C01743=-16.662,-86.143,37.169,176.3239,-5.7975,-6670.9471
C01744=-18.041,-88.518,38.031,179.9182,-0.1571,-6671.5198
C01745=-19.458,-91.164,38.697,-178.4928,2.5231,-6672.0484
C01746=-21.221,-93.510,39.027,-177.6909,1.9849,-6672.7860
C01747=-24.227,-95.023,39.203,-178.2776,0.4750,-6674.3034
C01748=-28.112,-95.435,39.346,-178.7289,-0.0594,-6676.4132
C01749=-32.220,-94.603,39.491,-179.9530,-0.0151,-6678.8079
C01750=-36.266,-93.184,39.587,-179.9934,-0.0025,-6681.2653
C01751=-40.247,-91.535,39.587,-179.9935,-0.0029,-6683.7346
C01752=-44.111,-89.678,39.491,-179.9560,-0.0226,-6686.1917
C01753=-47.604,-87.360,39.346,-179.0591,-0.8569,-6688.5867
C01754=-50.060,-84.322,39.203,-179.1177,-1.5538,-6690.6966
C01755=-51.116,-81.128,39.027,-179.7705,-3.0349,-6692.2136
C01756=-50.704,-78.221,38.697,179.2808,-2.8489,-6692.9519
C01757=-49.835,-75.348,38.031,-179.9468,0.1689,-6693.4806
C01758=-49.130,-72.694,37.169,-178.4898,6.6859,-6694.0527
C01759=-49.058,-70.314,36.333,179.0727,19.5923,-6694.9034
C01760=-50.194,-67.954,35.726,158.7492,29.2297,-6696.4513
C01761=-53.078,-65.141,35.484,150.6424,26.8233,-6699.1737
C01762=-56.256,-62.380,35.473,150.4564,26.9203,-6702.0450
C01763=-59.399,-59.399,35.480,151.7261,28.2744,-6705.0000
C01764=-62.380,-56.256,35.473,153.0793,29.5434,-6707.9550
C01765=-65.141,-53.078,35.484,153.1760,29.3567,-6710.8263
C01766=-67.954,-50.194,35.726,150.7705,21.2516,-6713.5487
C01767=-70.314,-49.058,36.333,160.4077,0.9273,-6715.0966
C01768=-72.694,-49.130,37.169,173.3141,-1.5102,-6715.9473
C01769=-75.348,-49.835,38.031,179.8311,-0.0532,-6716.5194
C01770=-78.221,-50.704,38.697,-177.1511,0.7192,-6717.0481
C01771=-81.128,-51.116,39.027,-176.9651,-0.2295,-6717.7864
C01772=-84.322,-50.060,39.203,-178.4462,-0.8823,-6719.3034
C01773=-87.360,-47.604,39.346,-179.1431,-0.9409,-6721.4133
C01774=-89.678,-44.111,39.491,-179.9774,-0.0440,-6723.8083
C01775=-91.535,-40.247,39.587,-179.9971,-0.0065,-6726.2654
C01776=-93.184,-36.266,39.587,-179.9975,-0.0066,-6728.7347
C01777=-94.603,-32.220,39.491,-179.9849,-0.0470,-6731.1921
C01778=-95.435,-28.112,39.346,-179.9406,-1.2711,-6733.5868
C01779=-95.023,-24.227,39.203,179.5250,-1.7224,-6735.6966
C01780=-93.510,-21.221,39.027,178.0151,-2.3091,-6737.2140
C01781=-91.164,-19.458,38.697,177.4769,-1.5072,-6737.9516
C01782=-88.518,-18.041,38.031,-179.8429,0.0818,-6738.4802
C01783=-86.143,-16.662,37.169,-174.2025,3.6761,-6739.0529
C01784=-84.409,-15.030,36.333,-166.4914,14.7419,-6739.9036
C01785=-83.543,-12.558,35.726,-173.1188,33.8482,-6741.4514
C01786=-83.594,-8.530,35.484,177.6980,37.0634,-6744.1737
C01787=-83.888,-4.330,35.473,177.6109,37.2284,-6747.0452
C01788=-84.003,0.000,35.480,-179.9996,37.2585,-6750.0000
C01789=-83.888,4.330,35.473,-177.6115,37.2285,-6752.9548
C01790=-83.594,8.530,35.484,-177.6995,37.0633,-6755.8263
C01791=-83.543,12.558,35.726,173.1197,33.8485,-6758.5486
C01792=-84.409,15.030,36.333,166.4914,14.7419,-6760.0964
C01793=-86.143,16.662,37.169,174.2025,3.6761,-6760.9471
C01794=-88.518,18.041,38.031,179.8429,0.0818,-6761.5198
C01795=-91.164,19.458,38.697,-177.4769,-1.5072,-6762.0484
C01796=-93.510,21.221,39.027,-178.0151,-2.3091,-6762.7860
C01797=-95.023,24.227,39.203,-179.5250,-1.7224,-6764.3034
C01798=-95.435,28.112,39.346,179.9406,-1.2711,-6766.4132
C01799=-94.603,32.220,39.491,179.9849,-0.0470,-6768.8079
C01800=-93.184,36.266,39.587,179.9975,-0.0066,-6771.2653
C01801=-91.535,40.247,39.587,179.9971,-0.0065,-6773.7346
C01802=-89.678,44.111,39.491,179.9774,-0.0440,-6776.1917
C01803=-87.360,47.604,39.346,179.1431,-0.9409,-6778.5867
C01804=-84.322,50.060,39.203,178.4462,-0.8823,-6780.6966
C01805=-81.128,51.116,39.027,176.9651,-0.2295,-6782.2136
C01806=-78.221,50.704,38.697,177.1511,0.7192,-6782.9519
C01807=-75.348,49.835,38.031,-179.8311,-0.0532,-6783.4806
C01808=-72.694,49.130,37.169,-173.3141,-1.5102,-6784.0527
C01809=-70.314,49.058,36.333,-160.4077,0.9273,-6784.9034
C01810=-67.954,50.194,35.726,-150.7703,21.2508,-6786.4513
C01811=-65.141,53.078,35.484,-153.1767,29.3576,-6789.1737
C01812=-62.380,56.256,35.473,-153.0797,29.5436,-6792.0450
C01813=-59.399,59.399,35.480,-151.7256,28.2739,-6795.0000
C01814=-56.256,62.380,35.473,-150.4566,26.9207,-6797.9550
C01815=-53.078,65.141,35.484,-150.6433,26.8240,-6800.8263
C01816=-50.194,67.954,35.726,-158.7484,29.2295,-6803.5487
C01817=-49.058,70.314,36.333,-179.0727,19.5923,-6805.0966
C01818=-49.130,72.694,37.169,178.4898,6.6859,-6805.9473
C01819=-49.835,75.348,38.031,179.9468,0.1689,-6806.5194
C01820=-50.704,78.221,38.697,-179.2808,-2.8489,-6807.0481
C01821=-51.116,81.128,39.027,179.7705,-3.0349,-6807.7864
C01822=-50.060,84.322,39.203,179.1177,-1.5538,-6809.3034
C01823=-47.604,87.360,39.346,179.0591,-0.8569,-6811.4133
C01824=-44.111,89.678,39.491,179.9560,-0.0226,-6813.8083
C01825=-40.247,91.535,39.587,179.9935,-0.0029,-6816.2654
C01826=-36.266,93.184,39.587,179.9934,-0.0025,-6818.7347
C01827=-32.220,94.603,39.491,179.9530,-0.0151,-6821.1921
C01828=-28.112,95.435,39.346,178.7289,-0.0594,-6823.5868
C01829=-24.227,95.023,39.203,178.2776,0.4750,-6825.6966
C01830=-21.221,93.510,39.027,177.6909,1.9849,-6827.2140
C01831=-19.458,91.164,38.697,178.4928,2.5231,-6827.9516
C01832=-18.041,88.518,38.031,-179.9182,-0.1571,-6828.4802
C01833=-16.662,86.143,37.169,-176.3239,-5.7975,-6829.0529
C01834=-15.030,84.409,36.333,-165.2581,-13.5086,-6829.9036
C01835=-12.558,83.543,35.726,-146.1515,-6.8803,-6831.4514
C01836=-8.530,83.594,35.484,-142.9367,2.3005,-6834.1737
C01837=-4.330,83.888,35.473,-142.7715,2.3885,-6837.0452
C01838=0.000,84.003,35.480,-142.7415,0.0004,-6840.0000
C01839=0.000,82.662,37.225,-142.2055,0.0004,-6840.0000
C01840=4.208,82.553,37.217,-142.2354,-2.4196,-6842.9180
C01841=8.324,82.270,37.229,-142.4103,-2.0928,-6845.7775
C01842=12.305,82.260,37.495,-146.1454,8.1058,-6848.5076
C01843=14.718,83.232,38.165,-167.2077,13.2282,-6850.0280
C01844=16.299,85.134,39.090,-177.2970,4.7574,-6850.8382
C01845=17.640,87.735,40.048,179.6311,-0.7865,-6851.3683
C01846=19.021,90.644,40.789,178.1721,-3.4318,-6851.8512
C01847=20.743,93.250,41.159,177.1705,-2.7402,-6852.5410
C01848=23.775,94.968,41.355,177.8447,-0.6817,-6854.0550
C01849=27.752,95.500,41.515,178.5424,0.0427,-6856.2037
C01850=31.992,94.679,41.678,179.9379,0.0198,-6858.6701
C01851=36.189,93.214,41.785,179.9917,0.0032,-6861.2180
C01852=40.323,91.502,41.785,179.9919,0.0036,-6863.7821
C01853=44.326,89.570,41.678,179.9421,0.0299,-6866.3297
C01854=47.905,87.153,41.515,178.9390,1.0006,-6868.7961
C01855=50.341,83.964,41.355,178.9574,2.0060,-6870.9450
C01856=51.270,80.606,41.159,179.9367,3.9353,-6872.4587
C01857=50.645,77.545,40.789,-178.8635,3.7173,-6873.1487
C01858=49.565,74.511,40.048,-179.7046,0.8170,-6873.6320
C01859=48.673,71.724,39.090,178.5413,-5.2696,-6874.1614
C01860=48.447,69.261,38.165,179.6754,-18.0958,-6874.9722
C01861=49.465,66.868,37.495,-159.5127,-29.9012,-6876.4919
C01862=52.288,64.059,37.229,-150.3090,-27.4069,-6879.2230
C01863=55.398,61.349,37.217,-149.9864,-27.3801,-6882.0820
C01864=58.451,58.451,37.225,-151.2608,-28.7396,-6885.0000
C01865=61.349,55.398,37.217,-152.6195,-30.0134,-6887.9180
C01866=64.059,52.288,37.229,-152.5923,-29.6900,-6890.7770
C01867=66.868,49.465,37.495,-150.0991,-20.4882,-6893.5081
C01868=69.261,48.447,38.165,-161.9042,0.3246,-6895.0278
C01869=71.724,48.673,39.090,-174.7304,1.4587,-6895.8386
C01870=74.511,49.565,40.048,179.1830,-0.2954,-6896.3680
C01871=77.545,50.645,40.789,176.2827,-1.1365,-6896.8513
C01872=80.606,51.270,41.159,176.0647,0.0633,-6897.5413
C01873=83.964,50.341,41.355,177.9940,1.0426,-6899.0550
C01874=87.153,47.905,41.515,178.9994,1.0610,-6901.2039
C01875=89.570,44.326,41.678,179.9701,0.0579,-6903.6703
C01876=91.502,40.323,41.785,179.9964,0.0081,-6906.2179
C01877=93.214,36.189,41.785,179.9968,0.0083,-6908.7820
C01878=94.679,31.992,41.678,179.9802,0.0621,-6911.3299
C01879=95.500,27.752,41.515,179.9573,1.4576,-6913.7963
C01880=94.968,23.775,41.355,-179.3183,2.1553,-6915.9450
C01881=93.250,20.743,41.159,-177.2598,2.8295,-6917.4590
C01882=90.644,19.021,40.789,-176.5682,1.8279,-6918.1488
C01883=87.735,17.640,40.048,-179.2135,0.3689,-6918.6317
C01884=85.134,16.299,39.090,175.2426,-2.7030,-6919.1618
C01885=83.232,14.718,38.165,166.7718,-12.7923,-6919.9720
C01886=82.260,12.305,37.495,171.8942,-33.8546,-6921.4924
C01887=82.270,8.324,37.229,-177.9072,-37.5897,-6924.2225
C01888=82.553,4.208,37.217,-177.5804,-37.7646,-6927.0820
C01889=82.662,0.000,37.225,179.9996,-37.7945,-6930.0000
C01890=82.553,-4.208,37.217,177.5810,-37.7647,-6932.9180
C01891=82.270,-8.324,37.229,177.9089,-37.5895,-6935.7775
C01892=82.260,-12.305,37.495,-171.8950,-33.8549,-6938.5076
C01893=83.232,-14.718,38.165,-166.7718,-12.7923,-6940.0280
C01894=85.134,-16.299,39.090,-175.2426,-2.7030,-6940.8382
C01895=87.735,-17.640,40.048,179.2135,0.3689,-6941.3683
C01896=90.644,-19.021,40.789,176.5682,1.8279,-6941.8512
C01897=93.250,-20.743,41.159,177.2598,2.8295,-6942.5410
C01898=94.968,-23.775,41.355,179.3183,2.1553,-6944.0550
C01899=95.500,-27.752,41.515,-179.9573,1.4576,-6946.2037
C01900=94.679,-31.992,41.678,-179.9802,0.0621,-6948.6701
C01901=93.214,-36.189,41.785,-179.9968,0.0083,-6951.2180
C01902=91.502,-40.323,41.785,-179.9964,0.0081,-6953.7821
C01903=89.570,-44.326,41.678,-179.9701,0.0579,-6956.3297
C01904=87.153,-47.905,41.515,-178.9994,1.0610,-6958.7961
C01905=83.964,-50.341,41.355,-177.9940,1.0426,-6960.9450
C01906=80.606,-51.270,41.159,-176.0647,0.0633,-6962.4587
C01907=77.545,-50.645,40.789,-176.2827,-1.1365,-6963.1487
C01908=74.511,-49.565,40.048,-179.1830,-0.2954,-6963.6320
C01909=71.724,-48.673,39.090,174.7304,1.4587,-6964.1614
C01910=69.261,-48.447,38.165,161.9042,0.3246,-6964.9722
C01911=66.868,-49.465,37.495,150.0988,-20.4873,-6966.4919
C01912=64.059,-52.288,37.229,152.5931,-29.6910,-6969.2230
C01913=61.349,-55.398,37.217,152.6199,-30.0136,-6972.0820
C01914=58.451,-58.451,37.225,151.2604,-28.7392,-6975.0000
C01915=55.398,-61.349,37.217,149.9866,-27.3805,-6977.9180
C01916=52.288,-64.059,37.229,150.3100,-27.4077,-6980.7770
C01917=49.465,-66.868,37.495,159.5118,-29.9009,-6983.5081
C01918=48.447,-69.261,38.165,-179.6754,-18.0958,-6985.0278
C01919=48.673,-71.724,39.090,-178.5413,-5.2696,-6985.8386
C01920=49.565,-74.511,40.048,179.7046,0.8170,-6986.3680
C01921=50.645,-77.545,40.789,178.8635,3.7173,-6986.8513
C01922=51.270,-80.606,41.159,-179.9367,3.9353,-6987.5413
C01923=50.341,-83.964,41.355,-178.9574,2.0060,-6989.0550
C01924=47.905,-87.153,41.515,-178.9390,1.0006,-6991.2039
C01925=44.326,-89.570,41.678,-179.9421,0.0299,-6993.6703
C01926=40.323,-91.502,41.785,-179.9919,0.0036,-6996.2179
C01927=36.189,-93.214,41.785,-179.9917,0.0032,-6998.7820
C01928=31.992,-94.679,41.678,-179.9379,0.0198,-7001.3299
C01929=27.752,-95.500,41.515,-178.5424,0.0427,-7003.7963
C01930=23.775,-94.968,41.355,-177.8447,-0.6817,-7005.9450
C01931=20.743,-93.250,41.159,-177.1705,-2.7402,-7007.4590
C01932=19.021,-90.644,40.789,-178.1721,-3.4318,-7008.1488
C01933=17.640,-87.735,40.048,-179.6311,-0.7865,-7008.6317
C01934=16.299,-85.134,39.090,177.2970,4.7574,-7009.1618
C01935=14.718,-83.232,38.165,167.2077,13.2282,-7009.9720
C01936=12.305,-82.260,37.495,146.1454,8.1058,-7011.4924
C01937=8.324,-82.270,37.229,142.4103,-2.0928,-7014.2225
C01938=4.208,-82.553,37.217,142.2354,-2.4196,-7017.0820
C01939=0.000,-82.662,37.225,142.2055,0.0004,-7020.0000
C01940=0.000,-82.662,37.225,142.2055,0.0004,-7020.0000
C01941=-4.208,-82.553,37.217,142.2353,2.4190,-7022.9180
C01942=-8.324,-82.270,37.229,142.4105,2.0911,-7025.7775
C01943=-12.305,-82.260,37.495,146.1451,-8.1050,-7028.5076
C01944=-14.718,-83.232,38.165,167.2077,-13.2282,-7030.0280
C01945=-16.299,-85.134,39.090,177.2970,-4.7574,-7030.8382
C01946=-17.640,-87.735,40.048,-179.6311,0.7865,-7031.3683
C01947=-19.021,-90.644,40.789,-178.1721,3.4318,-7031.8512
C01948=-20.743,-93.250,41.159,-177.1705,2.7402,-7032.5410
C01949=-23.775,-94.968,41.355,-177.8447,0.6817,-7034.0550
C01950=-27.752,-95.500,41.515,-178.5424,-0.0427,-7036.2037
C01951=-31.992,-94.679,41.678,-179.9379,-0.0198,-7038.6701
C01952=-36.189,-93.214,41.785,-179.9917,-0.0032,-7041.2180
C01953=-40.323,-91.502,41.785,-179.9919,-0.0036,-7043.7821
C01954=-44.326,-89.570,41.678,-179.9421,-0.0299,-7046.3297
C01955=-47.905,-87.153,41.515,-178.9390,-1.0006,-7048.7961
C01956=-50.341,-83.964,41.355,-178.9574,-2.0060,-7050.9450
C01957=-51.270,-80.606,41.159,-179.9367,-3.9353,-7052.4587
C01958=-50.645,-77.545,40.789,178.8635,-3.7173,-7053.1487
C01959=-49.565,-74.511,40.048,179.7046,-0.8170,-7053.6320
C01960=-48.673,-71.724,39.090,-178.5413,5.2696,-7054.1614
C01961=-48.447,-69.261,38.165,-179.6754,18.0958,-7054.9722
C01962=-49.465,-66.868,37.495,159.5127,29.9012,-7056.4919
C01963=-52.288,-64.059,37.229,150.3090,27.4069,-7059.2230
C01964=-55.398,-61.349,37.217,149.9864,27.3801,-7062.0820
C01965=-58.451,-58.451,37.225,151.2608,28.7396,-7065.0000
C01966=-61.349,-55.398,37.217,152.6195,30.0134,-7067.9180
C01967=-64.059,-52.288,37.229,152.5923,29.6900,-7070.7770
C01968=-66.868,-49.465,37.495,150.0991,20.4882,-7073.5081
C01969=-69.261,-48.447,38.165,161.9042,-0.3246,-7075.0278
C01970=-71.724,-48.673,39.090,174.7304,-1.4587,-7075.8386
C01971=-74.511,-49.565,40.048,-179.1830,0.2954,-7076.3680
C01972=-77.545,-50.645,40.789,-176.2827,1.1365,-7076.8513
C01973=-80.606,-51.270,41.159,-176.0647,-0.0633,-7077.5413
C01974=-83.964,-50.341,41.355,-177.9940,-1.0426,-7079.0550
C01975=-87.153,-47.905,41.515,-178.9994,-1.0610,-7081.2039
C01976=-89.570,-44.326,41.678,-179.9701,-0.0579,-7083.6703
C01977=-91.502,-40.323,41.785,-179.9964,-0.0081,-7086.2179
C01978=-93.214,-36.189,41.785,-179.9968,-0.0083,-7088.7820
C01979=-94.679,-31.992,41.678,-179.9802,-0.0621,-7091.3299
C01980=-95.500,-27.752,41.515,-179.9573,-1.4576,-7093.7963
C01981=-94.968,-23.775,41.355,179.3183,-2.1553,-7095.9450
C01982=-93.250,-20.743,41.159,177.2598,-2.8295,-7097.4590
C01983=-90.644,-19.021,40.789,176.5682,-1.8279,-7098.1488
C01984=-87.735,-17.640,40.048,179.2135,-0.3689,-7098.6317
C01985=-85.134,-16.299,39.090,-175.2426,2.7030,-7099.1618
C01986=-83.232,-14.718,38.165,-166.7718,12.7923,-7099.9720
C01987=-82.260,-12.305,37.495,-171.8942,33.8546,-7101.4924
C01988=-82.270,-8.324,37.229,177.9072,37.5897,-7104.2225
C01989=-82.553,-4.208,37.217,177.5804,37.7646,-7107.0820
C01990=-82.662,0.000,37.225,-179.9996,37.7945,-7110.0000
C01991=-82.553,4.208,37.217,-177.5810,37.7647,-7112.9180
C01992=-82.270,8.324,37.229,-177.9089,37.5895,-7115.7775
C01993=-82.260,12.305,37.495,171.8950,33.8549,-7118.5076
C01994=-83.232,14.718,38.165,166.7718,12.7923,-7120.0280
C01995=-85.134,16.299,39.090,175.2426,2.7030,-7120.8382
C01996=-87.735,17.640,40.048,-179.2135,-0.3689,-7121.3683
C01997=-90.644,19.021,40.789,-176.5682,-1.8279,-7121.8512
C01998=-93.250,20.743,41.159,-177.2598,-2.8295,-7122.5410
C01999=-94.968,23.775,41.355,-179.3183,-2.1553,-7124.0550
///TOOL 0
///POSTYPE ANGLE
///ANGLE
EC00000=0.0000,3566.7249
EC00001=0.0000,3567.6170
EC00002=0.0000,3568.5035
EC00003=0.0000,3569.6330
EC00004=0.0000,3571.2065
EC00005=0.0000,3573.0322
EC00006=0.0000,3574.8747
EC00007=0.0000,3576.6340
EC00008=0.0000,3578.3657
EC00009=0.0000,3580.1252
EC00010=0.0000,3581.9676
EC00011=0.0000,3583.7937
EC00012=0.0000,3585.3667
EC00013=0.0000,3586.4965
EC00014=0.0000,3587.3831
EC00015=0.0000,3588.2747
EC00016=0.0000,3589.4181
EC00017=0.0000,3591.1629
EC00018=0.0000,3593.8301
EC00019=0.0000,3596.7848
EC00020=0.0000,3600.0000
EC00021=0.0000,3600.0000
EC00022=0.0000,3603.1930
EC00023=0.0000,3606.1402
EC00024=0.0000,3608.8129
EC00025=0.0000,3610.5402
EC00026=0.0000,3611.6582
EC00027=0.0000,3612.5225
EC00028=0.0000,3613.3766
EC00029=0.0000,3614.4702
EC00030=0.0000,3616.0363
EC00031=0.0000,3617.8866
EC00032=0.0000,3619.7782
EC00033=0.0000,3621.6011
EC00034=0.0000,3623.3991
EC00035=0.0000,3625.2213
EC00036=0.0000,3627.1138
EC00037=0.0000,3628.9637
EC00038=0.0000,3630.5297
EC00039=0.0000,3631.6234
EC00040=0.0000,3632.4779
EC00041=0.0000,3633.3415
EC00042=0.0000,3634.4600
EC00043=0.0000,3636.1873
EC00044=0.0000,3638.8598
EC00045=0.0000,3641.8071
EC00046=0.0000,3645.0000
EC00047=0.0000,3648.1929
EC00048=0.0000,3651.1402
EC00049=0.0000,3653.8127
EC00050=0.0000,3655.5400
EC00051=0.0000,3656.6585
EC00052=0.0000,3657.5221
EC00053=0.0000,3658.3766
EC00054=0.0000,3659.4703
EC00055=0.0000,3661.0363
EC00056=0.0000,3662.8862
EC00057=0.0000,3664.7787
EC00058=0.0000,3666.6009
EC00059=0.0000,3668.3989
EC00060=0.0000,3670.2218
EC00061=0.0000,3672.1134
EC00062=0.0000,3673.9637
EC00063=0.0000,3675.5298
EC00064=0.0000,3676.6234
EC00065=0.0000,3677.4775
EC00066=0.0000,3678.3418
EC00067=0.0000,3679.4598
EC00068=0.0000,3681.1871
EC00069=0.0000,3683.8598
EC00070=0.0000,3686.8070
EC00071=0.0000,3690.0000
EC00072=0.0000,3693.1930
EC00073=0.0000,3696.1402
EC00074=0.0000,3698.8128
EC00075=0.0000,3700.5402
EC00076=0.0000,3701.6582
EC00077=0.0000,3702.5225
EC00078=0.0000,3703.3766
EC00079=0.0000,3704.4702
EC00080=0.0000,3706.0363
EC00081=0.0000,3707.8866
EC00082=0.0000,3709.7782
EC00083=0.0000,3711.6011
EC00084=0.0000,3713.3991
EC00085=0.0000,3715.2213
EC00086=0.0000,3717.1138
EC00087=0.0000,3718.9637
EC00088=0.0000,3720.5297
EC00089=0.0000,3721.6234
EC00090=0.0000,3722.4779
EC00091=0.0000,3723.3415
EC00092=0.0000,3724.4600
EC00093=0.0000,3726.1873
EC00094=0.0000,3728.8598
EC00095=0.0000,3731.8071
EC00096=0.0000,3735.0000
EC00097=0.0000,3738.1929
EC00098=0.0000,3741.1402
EC00099=0.0000,3743.8127
EC00100=0.0000,3745.5400
EC00101=0.0000,3746.6585
EC00102=0.0000,3747.5221
EC00103=0.0000,3748.3766
EC00104=0.0000,3749.4703
EC00105=0.0000,3751.0363
EC00106=0.0000,3752.8862
EC00107=0.0000,3754.7787
EC00108=0.0000,3756.6009
EC00109=0.0000,3758.3989
EC00110=0.0000,3760.2218
EC00111=0.0000,3762.1134
EC00112=0.0000,3763.9637
EC00113=0.0000,3765.5298
EC00114=0.0000,3766.6234
EC00115=0.0000,3767.4775
EC00116=0.0000,3768.3418
EC00117=0.0000,3769.4598
EC00118=0.0000,3771.1871
EC00119=0.0000,3773.8598
EC00120=0.0000,3776.8070
EC00121=0.0000,3780.0000
EC00122=0.0000,3780.0000
EC00123=0.0000,3783.1930
EC00124=0.0000,3786.1402
EC00125=0.0000,3788.8128
EC00126=0.0000,3790.5402
EC00127=0.0000,3791.6582
EC00128=0.0000,3792.5225
EC00129=0.0000,3793.3766
EC00130=0.0000,3794.4702
EC00131=0.0000,3796.0363
EC00132=0.0000,3797.8866
EC00133=0.0000,3799.7782
EC00134=0.0000,3801.6011
EC00135=0.0000,3803.3991
EC00136=0.0000,3805.2213
EC00137=0.0000,3807.1138
EC00138=0.0000,3808.9637
EC00139=0.0000,3810.5297
EC00140=0.0000,3811.6234
EC00141=0.0000,3812.4779
EC00142=0.0000,3813.3415
EC00143=0.0000,3814.4600
EC00144=0.0000,3816.1873
EC00145=0.0000,3818.8598
EC00146=0.0000,3821.8071
EC00147=0.0000,3825.0000
EC00148=0.0000,3828.1929
EC00149=0.0000,3831.1402
EC00150=0.0000,3833.8127
EC00151=0.0000,3835.5400
EC00152=0.0000,3836.6585
EC00153=0.0000,3837.5221
EC00154=0.0000,3838.3766
EC00155=0.0000,3839.4703
EC00156=0.0000,3841.0363
EC00157=0.0000,3842.8862
EC00158=0.0000,3844.7787
EC00159=0.0000,3846.6009
EC00160=0.0000,3848.3989
EC00161=0.0000,3850.2218
EC00162=0.0000,3852.1134
EC00163=0.0000,3853.9637
EC00164=0.0000,3855.5298
EC00165=0.0000,3856.6234
EC00166=0.0000,3857.4775
EC00167=0.0000,3858.3418
EC00168=0.0000,3859.4598
EC00169=0.0000,3861.1871
EC00170=0.0000,3863.8598
EC00171=0.0000,3866.8070
EC00172=0.0000,3870.0000
EC00173=0.0000,3873.1930
EC00174=0.0000,3876.1402
EC00175=0.0000,3878.8128
EC00176=0.0000,3880.5402
EC00177=0.0000,3881.6582
EC00178=0.0000,3882.5225
EC00179=0.0000,3883.3766
EC00180=0.0000,3884.4702
EC00181=0.0000,3886.0363
EC00182=0.0000,3887.8866
EC00183=0.0000,3889.7782
EC00184=0.0000,3891.6011
EC00185=0.0000,3893.3991
EC00186=0.0000,3895.2213
EC00187=0.0000,3897.1138
EC00188=0.0000,3898.9637
EC00189=0.0000,3900.5297
EC00190=0.0000,3901.6234
EC00191=0.0000,3902.4779
EC00192=0.0000,3903.3415
EC00193=0.0000,3904.4600
EC00194=0.0000,3906.1873
EC00195=0.0000,3908.8598
EC00196=0.0000,3911.8071
EC00197=0.0000,3915.0000
EC00198=0.0000,3918.1929
EC00199=0.0000,3921.1402
EC00200=0.0000,3923.8127
EC00201=0.0000,3925.5400
EC00202=0.0000,3926.6585
EC00203=0.0000,3927.5221
EC00204=0.0000,3928.3766
EC00205=0.0000,3929.4703
EC00206=0.0000,3931.0363
EC00207=0.0000,3932.8862
EC00208=0.0000,3934.7787
EC00209=0.0000,3936.6009
EC00210=0.0000,3938.3989
EC00211=0.0000,3940.2218
EC00212=0.0000,3942.1134
EC00213=0.0000,3943.9637
EC00214=0.0000,3945.5298
EC00215=0.0000,3946.6234
EC00216=0.0000,3947.4775
EC00217=0.0000,3948.3418
EC00218=0.0000,3949.4598
EC00219=0.0000,3951.1872
EC00220=0.0000,3953.8598
EC00221=0.0000,3956.8070
EC00222=0.0000,3960.0000
EC00223=0.0000,3960.0000
EC00224=0.0000,3963.1693
EC00225=0.0000,3966.1086
EC00226=0.0000,3968.7858
EC00227=0.0000,3970.4951
EC00228=0.0000,3971.5862
EC00229=0.0000,3972.4199
EC00230=0.0000,3973.2394
EC00231=0.0000,3974.2944
EC00232=0.0000,3975.8535
EC00233=0.0000,3977.7299
EC00234=0.0000,3979.6757
EC00235=0.0000,3981.5655
EC00236=0.0000,3983.4348
EC00237=0.0000,3985.3246
EC00238=0.0000,3987.2701
EC00239=0.0000,3989.1464
EC00240=0.0000,3990.7059
EC00241=0.0000,3991.7605
EC00242=0.0000,3992.5800
EC00243=0.0000,3993.4139
EC00244=0.0000,3994.5045
EC00245=0.0000,3996.2144
EC00246=0.0000,3998.8913
EC00247=0.0000,4001.8309
EC00248=0.0000,4005.0000
EC00249=0.0000,4008.1691
EC00250=0.0000,4011.1087
EC00251=0.0000,4013.7856
EC00252=0.0000,4015.4955
EC00253=0.0000,4016.5861
EC00254=0.0000,4017.4200
EC00255=0.0000,4018.2395
EC00256=0.0000,4019.2941
EC00257=0.0000,4020.8536
EC00258=0.0000,4022.7299
EC00259=0.0000,4024.6754
EC00260=0.0000,4026.5652
EC00261=0.0000,4028.4345
EC00262=0.0000,4030.3243
EC00263=0.0000,4032.2701
EC00264=0.0000,4034.1465
EC00265=0.0000,4035.7056
EC00266=0.0000,4036.7606
EC00267=0.0000,4037.5801
EC00268=0.0000,4038.4138
EC00269=0.0000,4039.5049
EC00270=0.0000,4041.2142
EC00271=0.0000,4043.8914
EC00272=0.0000,4046.8307
EC00273=0.0000,4050.0000
EC00274=0.0000,4053.1693
EC00275=0.0000,4056.1086
EC00276=0.0000,4058.7858
EC00277=0.0000,4060.4951
EC00278=0.0000,4061.5862
EC00279=0.0000,4062.4199
EC00280=0.0000,4063.2394
EC00281=0.0000,4064.2944
EC00282=0.0000,4065.8535
EC00283=0.0000,4067.7299
EC00284=0.0000,4069.6757
EC00285=0.0000,4071.5655
EC00286=0.0000,4073.4348
EC00287=0.0000,4075.3246
EC00288=0.0000,4077.2701
EC00289=0.0000,4079.1464
EC00290=0.0000,4080.7059
EC00291=0.0000,4081.7605
EC00292=0.0000,4082.5800
EC00293=0.0000,4083.4139
EC00294=0.0000,4084.5045
EC00295=0.0000,4086.2144
EC00296=0.0000,4088.8913
EC00297=0.0000,4091.8309
EC00298=0.0000,4095.0000
EC00299=0.0000,4098.1691
EC00300=0.0000,4101.1087
EC00301=0.0000,4103.7856
EC00302=0.0000,4105.4955
EC00303=0.0000,4106.5861
EC00304=0.0000,4107.4200
EC00305=0.0000,4108.2395
EC00306=0.0000,4109.2941
EC00307=0.0000,4110.8536
EC00308=0.0000,4112.7299
EC00309=0.0000,4114.6754
EC00310=0.0000,4116.5652
EC00311=0.0000,4118.4345
EC00312=0.0000,4120.3243
EC00313=0.0000,4122.2701
EC00314=0.0000,4124.1465
EC00315=0.0000,4125.7056
EC00316=0.0000,4126.7606
EC00317=0.0000,4127.5801
EC00318=0.0000,4128.4138
EC00319=0.0000,4129.5049
EC00320=0.0000,4131.2142
EC00321=0.0000,4133.8914
EC00322=0.0000,4136.8307
EC00323=0.0000,4140.0000
EC00324=0.0000,4140.0000
EC00325=0.0000,4143.1693
EC00326=0.0000,4146.1086
EC00327=0.0000,4148.7858
EC00328=0.0000,4150.4951
EC00329=0.0000,4151.5862
EC00330=0.0000,4152.4199
EC00331=0.0000,4153.2394
EC00332=0.0000,4154.2944
EC00333=0.0000,4155.8535
EC00334=0.0000,4157.7299
EC00335=0.0000,4159.6757
EC00336=0.0000,4161.5655
EC00337=0.0000,4163.4348
EC00338=0.0000,4165.3246
EC00339=0.0000,4167.2701
EC00340=0.0000,4169.1464
EC00341=0.0000,4170.7059
EC00342=0.0000,4171.7605
EC00343=0.0000,4172.5800
EC00344=0.0000,4173.4139
EC00345=0.0000,4174.5045
EC00346=0.0000,4176.2144
EC00347=0.0000,4178.8913
EC00348=0.0000,4181.8309
EC00349=0.0000,4185.0000
EC00350=0.0000,4188.1691
EC00351=0.0000,4191.1087
EC00352=0.0000,4193.7856
EC00353=0.0000,4195.4955
EC00354=0.0000,4196.5861
EC00355=0.0000,4197.4200
EC00356=0.0000,4198.2395
EC00357=0.0000,4199.2941
EC00358=0.0000,4200.8536
EC00359=0.0000,4202.7299
EC00360=0.0000,4204.6754
EC00361=0.0000,4206.5652
EC00362=0.0000,4208.4345
EC00363=0.0000,4210.3243
EC00364=0.0000,4212.2701
EC00365=0.0000,4214.1465
EC00366=0.0000,4215.7056
EC00367=0.0000,4216.7606
EC00368=0.0000,4217.5801
EC00369=0.0000,4218.4138
EC00370=0.0000,4219.5049
EC00371=0.0000,4221.2142
EC00372=0.0000,4223.8914
EC00373=0.0000,4226.8307
EC00374=0.0000,4230.0000
EC00375=0.0000,4233.1693
EC00376=0.0000,4236.1086
EC00377=0.0000,4238.7858
EC00378=0.0000,4240.4951
EC00379=0.0000,4241.5862
EC00380=0.0000,4242.4199
EC00381=0.0000,4243.2394
EC00382=0.0000,4244.2944
EC00383=0.0000,4245.8535
EC00384=0.0000,4247.7299
EC00385=0.0000,4249.6757
EC00386=0.0000,4251.5655
EC00387=0.0000,4253.4348
EC00388=0.0000,4255.3246
EC00389=0.0000,4257.2701
EC00390=0.0000,4259.1464
EC00391=0.0000,4260.7059
EC00392=0.0000,4261.7605
EC00393=0.0000,4262.5800
EC00394=0.0000,4263.4139
EC00395=0.0000,4264.5045
EC00396=0.0000,4266.2144
EC00397=0.0000,4268.8913
EC00398=0.0000,4271.8309
EC00399=0.0000,4275.0000
EC00400=0.0000,4278.1691
EC00401=0.0000,4281.1087
EC00402=0.0000,4283.7856
EC00403=0.0000,4285.4955
EC00404=0.0000,4286.5861
EC00405=0.0000,4287.4200
EC00406=0.0000,4288.2395
EC00407=0.0000,4289.2941
EC00408=0.0000,4290.8536
EC00409=0.0000,4292.7299
EC00410=0.0000,4294.6754
EC00411=0.0000,4296.5652
EC00412=0.0000,4298.4345
EC00413=0.0000,4300.3243
EC00414=0.0000,4302.2701
EC00415=0.0000,4304.1465
EC00416=0.0000,4305.7056
EC00417=0.0000,4306.7606
EC00418=0.0000,4307.5801
EC00419=0.0000,4308.4138
EC00420=0.0000,4309.5049
EC00421=0.0000,4311.2142
EC00422=0.0000,4313.8914
EC00423=0.0000,4316.8307
EC00424=0.0000,4320.0000
EC00425=0.0000,4320.0000
EC00426=0.0000,4323.1434
EC00427=0.0000,4326.0750
EC00428=0.0000,4328.7577
EC00429=0.0000,4330.4474
EC00430=0.0000,4331.5089
EC00431=0.0000,4332.3101
EC00432=0.0000,4333.0930
EC00433=0.0000,4334.1066
EC00434=0.0000,4335.6587
EC00435=0.0000,4337.5637
EC00436=0.0000,4339.5659
EC00437=0.0000,4341.5274
EC00438=0.0000,4343.4725
EC00439=0.0000,4345.4343
EC00440=0.0000,4347.4359
EC00441=0.0000,4349.3411
EC00442=0.0000,4350.8935
EC00443=0.0000,4351.9071
EC00444=0.0000,4352.6899
EC00445=0.0000,4353.4910
EC00446=0.0000,4354.5530
EC00447=0.0000,4356.2423
EC00448=0.0000,4358.9252
EC00449=0.0000,4361.8567
EC00450=0.0000,4365.0000
EC00451=0.0000,4368.1433
EC00452=0.0000,4371.0748
EC00453=0.0000,4373.7577
EC00454=0.0000,4375.4470
EC00455=0.0000,4376.5090
EC00456=0.0000,4377.3101
EC00457=0.0000,4378.0929
EC00458=0.0000,4379.1065
EC00459=0.0000,4380.6589
EC00460=0.0000,4382.5641
EC00461=0.0000,4384.5657
EC00462=0.0000,4386.5275
EC00463=0.0000,4388.4726
EC00464=0.0000,4390.4341
EC00465=0.0000,4392.4363
EC00466=0.0000,4394.3413
EC00467=0.0000,4395.8934
EC00468=0.0000,4396.9070
EC00469=0.0000,4397.6899
EC00470=0.0000,4398.4911
EC00471=0.0000,4399.5526
EC00472=0.0000,4401.2423
EC00473=0.0000,4403.9250
EC00474=0.0000,4406.8566
EC00475=0.0000,4410.0000
EC00476=0.0000,4413.1434
EC00477=0.0000,4416.0750
EC00478=0.0000,4418.7577
EC00479=0.0000,4420.4474
EC00480=0.0000,4421.5089
EC00481=0.0000,4422.3101
EC00482=0.0000,4423.0930
EC00483=0.0000,4424.1066
EC00484=0.0000,4425.6587
EC00485=0.0000,4427.5637
EC00486=0.0000,4429.5659
EC00487=0.0000,4431.5274
EC00488=0.0000,4433.4725
EC00489=0.0000,4435.4343
EC00490=0.0000,4437.4359
EC00491=0.0000,4439.3411
EC00492=0.0000,4440.8935
EC00493=0.0000,4441.9071
EC00494=0.0000,4442.6899
EC00495=0.0000,4443.4910
EC00496=0.0000,4444.5530
EC00497=0.0000,4446.2423
EC00498=0.0000,4448.9252
EC00499=0.0000,4451.8567
EC00500=0.0000,4455.0000
EC00501=0.0000,4458.1433
EC00502=0.0000,4461.0748
EC00503=0.0000,4463.7577
EC00504=0.0000,4465.4470
EC00505=0.0000,4466.5090
EC00506=0.0000,4467.3101
EC00507=0.0000,4468.0929
EC00508=0.0000,4469.1065
EC00509=0.0000,4470.6589
EC00510=0.0000,4472.5641
EC00511=0.0000,4474.5657
EC00512=0.0000,4476.5275
EC00513=0.0000,4478.4726
EC00514=0.0000,4480.4341
EC00515=0.0000,4482.4363
EC00516=0.0000,4484.3413
EC00517=0.0000,4485.8934
EC00518=0.0000,4486.9070
EC00519=0.0000,4487.6899
EC00520=0.0000,4488.4911
EC00521=0.0000,4489.5526
EC00522=0.0000,4491.2423
EC00523=0.0000,4493.9250
EC00524=0.0000,4496.8566
EC00525=0.0000,4500.0000
EC00526=0.0000,4500.0000
EC00527=0.0000,4503.1434
EC00528=0.0000,4506.0750
EC00529=0.0000,4508.7577
EC00530=0.0000,4510.4474
EC00531=0.0000,4511.5089
EC00532=0.0000,4512.3101
EC00533=0.0000,4513.0930
EC00534=0.0000,4514.1066
EC00535=0.0000,4515.6587
EC00536=0.0000,4517.5637
EC00537=0.0000,4519.5659
EC00538=0.0000,4521.5274
EC00539=0.0000,4523.4725
EC00540=0.0000,4525.4343
EC00541=0.0000,4527.4359
EC00542=0.0000,4529.3411
EC00543=0.0000,4530.8935
EC00544=0.0000,4531.9071
EC00545=0.0000,4532.6899
EC00546=0.0000,4533.4910
EC00547=0.0000,4534.5530
EC00548=0.0000,4536.2423
EC00549=0.0000,4538.9252
EC00550=0.0000,4541.8567
EC00551=0.0000,4545.0000
EC00552=0.0000,4548.1433
EC00553=0.0000,4551.0748
EC00554=0.0000,4553.7577
EC00555=0.0000,4555.4470
EC00556=0.0000,4556.5090
EC00557=0.0000,4557.3101
EC00558=0.0000,4558.0929
EC00559=0.0000,4559.1065
EC00560=0.0000,4560.6589
EC00561=0.0000,4562.5641
EC00562=0.0000,4564.5657
EC00563=0.0000,4566.5275
EC00564=0.0000,4568.4726
EC00565=0.0000,4570.4341
EC00566=0.0000,4572.4363
EC00567=0.0000,4574.3413
EC00568=0.0000,4575.8934
EC00569=0.0000,4576.9070
EC00570=0.0000,4577.6899
EC00571=0.0000,4578.4911
EC00572=0.0000,4579.5526
EC00573=0.0000,4581.2423
EC00574=0.0000,4583.9250
EC00575=0.0000,4586.8566
EC00576=0.0000,4590.0000
EC00577=0.0000,4593.1434
EC00578=0.0000,4596.0750
EC00579=0.0000,4598.7577
EC00580=0.0000,4600.4474
EC00581=0.0000,4601.5089
EC00582=0.0000,4602.3101
EC00583=0.0000,4603.0930
EC00584=0.0000,4604.1066
EC00585=0.0000,4605.6587
EC00586=0.0000,4607.5637
EC00587=0.0000,4609.5659
EC00588=0.0000,4611.5274
EC00589=0.0000,4613.4725
EC00590=0.0000,4615.4343
EC00591=0.0000,4617.4359
EC00592=0.0000,4619.3411
EC00593=0.0000,4620.8935
EC00594=0.0000,4621.9071
EC00595=0.0000,4622.6899
EC00596=0.0000,4623.4910
EC00597=0.0000,4624.5530
EC00598=0.0000,4626.2423
EC00599=0.0000,4628.9252
EC00600=0.0000,4631.8567
EC00601=0.0000,4635.0000
EC00602=0.0000,4638.1433
EC00603=0.0000,4641.0748
EC00604=0.0000,4643.7577
EC00605=0.0000,4645.4470
EC00606=0.0000,4646.5090
EC00607=0.0000,4647.3101
EC00608=0.0000,4648.0929
EC00609=0.0000,4649.1065
EC00610=0.0000,4650.6589
EC00611=0.0000,4652.5641
EC00612=0.0000,4654.5657
EC00613=0.0000,4656.5275
EC00614=0.0000,4658.4726
EC00615=0.0000,4660.4341
EC00616=0.0000,4662.4363
EC00617=0.0000,4664.3413
EC00618=0.0000,4665.8934
EC00619=0.0000,4666.9070
EC00620=0.0000,4667.6899
EC00621=0.0000,4668.4911
EC00622=0.0000,4669.5526
EC00623=0.0000,4671.2423
EC00624=0.0000,4673.9250
EC00625=0.0000,4676.8566
EC00626=0.0000,4680.0000
EC00627=0.0000,4680.0000
EC00628=0.0000,4683.1159
EC00629=0.0000,4686.0385
EC00630=0.0000,4688.7274
EC00631=0.0000,4690.3963
EC00632=0.0000,4691.4267
EC00633=0.0000,4692.1938
EC00634=0.0000,4692.9380
EC00635=0.0000,4693.9087
EC00636=0.0000,4695.4538
EC00637=0.0000,4697.3887
EC00638=0.0000,4699.4506
EC00639=0.0000,4701.4875
EC00640=0.0000,4703.5125
EC00641=0.0000,4705.5494
EC00642=0.0000,4707.6113
EC00643=0.0000,4709.5463
EC00644=0.0000,4711.0916
EC00645=0.0000,4712.0621
EC00646=0.0000,4712.8061
EC00647=0.0000,4713.5730
EC00648=0.0000,4714.6038
EC00649=0.0000,4716.2732
EC00650=0.0000,4718.9613
EC00651=0.0000,4721.8843
EC00652=0.0000,4725.0000
EC00653=0.0000,4728.1157
EC00654=0.0000,4731.0387
EC00655=0.0000,4733.7268
EC00656=0.0000,4735.3962
EC00657=0.0000,4736.4270
EC00658=0.0000,4737.1939
EC00659=0.0000,4737.9379
EC00660=0.0000,4738.9084
EC00661=0.0000,4740.4537
EC00662=0.0000,4742.3887
EC00663=0.0000,4744.4506
EC00664=0.0000,4746.4875
EC00665=0.0000,4748.5125
EC00666=0.0000,4750.5494
EC00667=0.0000,4752.6113
EC00668=0.0000,4754.5462
EC00669=0.0000,4756.0913
EC00670=0.0000,4757.0620
EC00671=0.0000,4757.8062
EC00672=0.0000,4758.5733
EC00673=0.0000,4759.6037
EC00674=0.0000,4761.2726
EC00675=0.0000,4763.9615
EC00676=0.0000,4766.8841
EC00677=0.0000,4770.0000
EC00678=0.0000,4773.1159
EC00679=0.0000,4776.0385
EC00680=0.0000,4778.7274
EC00681=0.0000,4780.3963
EC00682=0.0000,4781.4267
EC00683=0.0000,4782.1938
EC00684=0.0000,4782.9380
EC00685=0.0000,4783.9087
EC00686=0.0000,4785.4538
EC00687=0.0000,4787.3887
EC00688=0.0000,4789.4506
EC00689=0.0000,4791.4875
EC00690=0.0000,4793.5125
EC00691=0.0000,4795.5494
EC00692=0.0000,4797.6113
EC00693=0.0000,4799.5463
EC00694=0.0000,4801.0916
EC00695=0.0000,4802.0621
EC00696=0.0000,4802.8061
EC00697=0.0000,4803.5730
EC00698=0.0000,4804.6038
EC00699=0.0000,4806.2732
EC00700=0.0000,4808.9613
EC00701=0.0000,4811.8843
EC00702=0.0000,4815.0000
EC00703=0.0000,4818.1157
EC00704=0.0000,4821.0387
EC00705=0.0000,4823.7268
EC00706=0.0000,4825.3962
EC00707=0.0000,4826.4270
EC00708=0.0000,4827.1939
EC00709=0.0000,4827.9379
EC00710=0.0000,4828.9084
EC00711=0.0000,4830.4537
EC00712=0.0000,4832.3887
EC00713=0.0000,4834.4506
EC00714=0.0000,4836.4875
EC00715=0.0000,4838.5125
EC00716=0.0000,4840.5494
EC00717=0.0000,4842.6113
EC00718=0.0000,4844.5462
EC00719=0.0000,4846.0913
EC00720=0.0000,4847.0620
EC00721=0.0000,4847.8062
EC00722=0.0000,4848.5733
EC00723=0.0000,4849.6037
EC00724=0.0000,4851.2726
EC00725=0.0000,4853.9615
EC00726=0.0000,4856.8841
EC00727=0.0000,4860.0000
EC00728=0.0000,4860.0000
EC00729=0.0000,4863.1159
EC00730=0.0000,4866.0385
EC00731=0.0000,4868.7274
EC00732=0.0000,4870.3963
EC00733=0.0000,4871.4267
EC00734=0.0000,4872.1938
EC00735=0.0000,4872.9380
EC00736=0.0000,4873.9087
EC00737=0.0000,4875.4538
EC00738=0.0000,4877.3887
EC00739=0.0000,4879.4506
EC00740=0.0000,4881.4875
EC00741=0.0000,4883.5125
EC00742=0.0000,4885.5494
EC00743=0.0000,4887.6113
EC00744=0.0000,4889.5463
EC00745=0.0000,4891.0916
EC00746=0.0000,4892.0621
EC00747=0.0000,4892.8061
EC00748=0.0000,4893.5730
EC00749=0.0000,4894.6038
EC00750=0.0000,4896.2732
EC00751=0.0000,4898.9613
EC00752=0.0000,4901.8843
EC00753=0.0000,4905.0000
EC00754=0.0000,4908.1157
EC00755=0.0000,4911.0387
EC00756=0.0000,4913.7268
EC00757=0.0000,4915.3962
EC00758=0.0000,4916.4270
EC00759=0.0000,4917.1939
EC00760=0.0000,4917.9379
EC00761=0.0000,4918.9084
EC00762=0.0000,4920.4537
EC00763=0.0000,4922.3887
EC00764=0.0000,4924.4506
EC00765=0.0000,4926.4875
EC00766=0.0000,4928.5125
EC00767=0.0000,4930.5494
EC00768=0.0000,4932.6113
EC00769=0.0000,4934.5462
EC00770=0.0000,4936.0913
EC00771=0.0000,4937.0620
EC00772=0.0000,4937.8062
EC00773=0.0000,4938.5733
EC00774=0.0000,4939.6037
EC00775=0.0000,4941.2726
EC00776=0.0000,4943.9615
EC00777=0.0000,4946.8841
EC00778=0.0000,4950.0000
EC00779=0.0000,4953.1159
EC00780=0.0000,4956.0385
EC00781=0.0000,4958.7274
EC00782=0.0000,4960.3963
EC00783=0.0000,4961.4267
EC00784=0.0000,4962.1938
EC00785=0.0000,4962.9380
EC00786=0.0000,4963.9087
EC00787=0.0000,4965.4538
EC00788=0.0000,4967.3887
EC00789=0.0000,4969.4506
EC00790=0.0000,4971.4875
EC00791=0.0000,4973.5125
EC00792=0.0000,4975.5494
EC00793=0.0000,4977.6113
EC00794=0.0000,4979.5463
EC00795=0.0000,4981.0916
EC00796=0.0000,4982.0621
EC00797=0.0000,4982.8061
EC00798=0.0000,4983.5730
EC00799=0.0000,4984.6038
EC00800=0.0000,4986.2732
EC00801=0.0000,4988.9613
EC00802=0.0000,4991.8843
EC00803=0.0000,4995.0000
EC00804=0.0000,4998.1157
EC00805=0.0000,5001.0387
EC00806=0.0000,5003.7268
EC00807=0.0000,5005.3962
EC00808=0.0000,5006.4270
EC00809=0.0000,5007.1939
EC00810=0.0000,5007.9379
EC00811=0.0000,5008.9084
EC00812=0.0000,5010.4537
EC00813=0.0000,5012.3887
EC00814=0.0000,5014.4506
EC00815=0.0000,5016.4875
EC00816=0.0000,5018.5125
EC00817=0.0000,5020.5494
EC00818=0.0000,5022.6113
EC00819=0.0000,5024.5462
EC00820=0.0000,5026.0913
EC00821=0.0000,5027.0620
EC00822=0.0000,5027.8062
EC00823=0.0000,5028.5733
EC00824=0.0000,5029.6037
EC00825=0.0000,5031.2726
EC00826=0.0000,5033.9615
EC00827=0.0000,5036.8841
EC00828=0.0000,5040.0000
EC00829=0.0000,5040.0000
EC00830=0.0000,5043.0871
EC00831=0.0000,5046.0002
EC00832=0.0000,5048.6952
EC00833=0.0000,5050.3419
EC00834=0.0000,5051.3400
EC00835=0.0000,5052.0705
EC00836=0.0000,5052.7745
EC00837=0.0000,5053.7009
EC00838=0.0000,5055.2391
EC00839=0.0000,5057.2060
EC00840=0.0000,5059.3299
EC00841=0.0000,5061.4458
EC00842=0.0000,5063.5540
EC00843=0.0000,5065.6698
EC00844=0.0000,5067.7938
EC00845=0.0000,5069.7609
EC00846=0.0000,5071.2994
EC00847=0.0000,5072.2255
EC00848=0.0000,5072.9290
EC00849=0.0000,5073.6599
EC00850=0.0000,5074.6583
EC00851=0.0000,5076.3048
EC00852=0.0000,5078.9993
EC00853=0.0000,5081.9128
EC00854=0.0000,5085.0000
EC00855=0.0000,5088.0872
EC00856=0.0000,5091.0007
EC00857=0.0000,5093.6952
EC00858=0.0000,5095.3417
EC00859=0.0000,5096.3401
EC00860=0.0000,5097.0710
EC00861=0.0000,5097.7745
EC00862=0.0000,5098.7006
EC00863=0.0000,5100.2391
EC00864=0.0000,5102.2062
EC00865=0.0000,5104.3302
EC00866=0.0000,5106.4460
EC00867=0.0000,5108.5542
EC00868=0.0000,5110.6701
EC00869=0.0000,5112.7940
EC00870=0.0000,5114.7609
EC00871=0.0000,5116.2991
EC00872=0.0000,5117.2255
EC00873=0.0000,5117.9295
EC00874=0.0000,5118.6600
EC00875=0.0000,5119.6581
EC00876=0.0000,5121.3048
EC00877=0.0000,5123.9998
EC00878=0.0000,5126.9129
EC00879=0.0000,5130.0000
EC00880=0.0000,5133.0871
EC00881=0.0000,5136.0002
EC00882=0.0000,5138.6952
EC00883=0.0000,5140.3419
EC00884=0.0000,5141.3400
EC00885=0.0000,5142.0705
EC00886=0.0000,5142.7745
EC00887=0.0000,5143.7009
EC00888=0.0000,5145.2391
EC00889=0.0000,5147.2060
EC00890=0.0000,5149.3299
EC00891=0.0000,5151.4458
EC00892=0.0000,5153.5540
EC00893=0.0000,5155.6698
EC00894=0.0000,5157.7938
EC00895=0.0000,5159.7609
EC00896=0.0000,5161.2994
EC00897=0.0000,5162.2255
EC00898=0.0000,5162.9290
EC00899=0.0000,5163.6599
EC00900=0.0000,5164.6583
EC00901=0.0000,5166.3048
EC00902=0.0000,5168.9993
EC00903=0.0000,5171.9128
EC00904=0.0000,5175.0000
EC00905=0.0000,5178.0872
EC00906=0.0000,5181.0007
EC00907=0.0000,5183.6952
EC00908=0.0000,5185.3417
EC00909=0.0000,5186.3401
EC00910=0.0000,5187.0710
EC00911=0.0000,5187.7745
EC00912=0.0000,5188.7006
EC00913=0.0000,5190.2391
EC00914=0.0000,5192.2062
EC00915=0.0000,5194.3302
EC00916=0.0000,5196.4460
EC00917=0.0000,5198.5542
EC00918=0.0000,5200.6701
EC00919=0.0000,5202.7940
EC00920=0.0000,5204.7609
EC00921=0.0000,5206.2991
EC00922=0.0000,5207.2255
EC00923=0.0000,5207.9295
EC00924=0.0000,5208.6600
EC00925=0.0000,5209.6581
EC00926=0.0000,5211.3048
EC00927=0.0000,5213.9998
EC00928=0.0000,5216.9129
EC00929=0.0000,5220.0000
EC00930=0.0000,5220.0000
EC00931=0.0000,5223.0871
EC00932=0.0000,5226.0002
EC00933=0.0000,5228.6952
EC00934=0.0000,5230.3419
EC00935=0.0000,5231.3400
EC00936=0.0000,5232.0705
EC00937=0.0000,5232.7745
EC00938=0.0000,5233.7009
EC00939=0.0000,5235.2391
EC00940=0.0000,5237.2060
EC00941=0.0000,5239.3299
EC00942=0.0000,5241.4458
EC00943=0.0000,5243.5540
EC00944=0.0000,5245.6698
EC00945=0.0000,5247.7938
EC00946=0.0000,5249.7609
EC00947=0.0000,5251.2994
EC00948=0.0000,5252.2255
EC00949=0.0000,5252.9290
EC00950=0.0000,5253.6599
EC00951=0.0000,5254.6583
EC00952=0.0000,5256.3048
EC00953=0.0000,5258.9993
EC00954=0.0000,5261.9128
EC00955=0.0000,5265.0000
EC00956=0.0000,5268.0872
EC00957=0.0000,5271.0007
EC00958=0.0000,5273.6952
EC00959=0.0000,5275.3417
EC00960=0.0000,5276.3401
EC00961=0.0000,5277.0710
EC00962=0.0000,5277.7745
EC00963=0.0000,5278.7006
EC00964=0.0000,5280.2391
EC00965=0.0000,5282.2062
EC00966=0.0000,5284.3302
EC00967=0.0000,5286.4460
EC00968=0.0000,5288.5542
EC00969=0.0000,5290.6701
EC00970=0.0000,5292.7940
EC00971=0.0000,5294.7609
EC00972=0.0000,5296.2991
EC00973=0.0000,5297.2255
EC00974=0.0000,5297.9295
EC00975=0.0000,5298.6600
EC00976=0.0000,5299.6581
EC00977=0.0000,5301.3048
EC00978=0.0000,5303.9998
EC00979=0.0000,5306.9129
EC00980=0.0000,5310.0000
EC00981=0.0000,5313.0871
EC00982=0.0000,5316.0002
EC00983=0.0000,5318.6952
EC00984=0.0000,5320.3419
EC00985=0.0000,5321.3400
EC00986=0.0000,5322.0705
EC00987=0.0000,5322.7745
EC00988=0.0000,5323.7009
EC00989=0.0000,5325.2391
EC00990=0.0000,5327.2060
EC00991=0.0000,5329.3299
EC00992=0.0000,5331.4458
EC00993=0.0000,5333.5540
EC00994=0.0000,5335.6698
EC00995=0.0000,5337.7938
EC00996=0.0000,5339.7609
EC00997=0.0000,5341.2994
EC00998=0.0000,5342.2255
EC00999=0.0000,5342.9290
EC01000=0.0000,5343.6599
EC01001=0.0000,5344.6583
EC01002=0.0000,5346.3048
EC01003=0.0000,5348.9993
EC01004=0.0000,5351.9128
EC01005=0.0000,5355.0000
EC01006=0.0000,5358.0872
EC01007=0.0000,5361.0007
EC01008=0.0000,5363.6952
EC01009=0.0000,5365.3417
EC01010=0.0000,5366.3401
EC01011=0.0000,5367.0710
EC01012=0.0000,5367.7745
EC01013=0.0000,5368.7006
EC01014=0.0000,5370.2391
EC01015=0.0000,5372.2062
EC01016=0.0000,5374.3302
EC01017=0.0000,5376.4460
EC01018=0.0000,5378.5542
EC01019=0.0000,5380.6701
EC01020=0.0000,5382.7940
EC01021=0.0000,5384.7609
EC01022=0.0000,5386.2991
EC01023=0.0000,5387.2255
EC01024=0.0000,5387.9295
EC01025=0.0000,5388.6600
EC01026=0.0000,5389.6581
EC01027=0.0000,5391.3048
EC01028=0.0000,5393.9998
EC01029=0.0000,5396.9129
EC01030=0.0000,5400.0000
EC01031=0.0000,5400.0000
EC01032=0.0000,5403.0565
EC01033=0.0000,5405.9598
EC01034=0.0000,5408.6610
EC01035=0.0000,5410.2852
EC01036=0.0000,5411.2483
EC01037=0.0000,5411.9417
EC01038=0.0000,5412.6030
EC01039=0.0000,5413.4837
EC01040=0.0000,5415.0155
EC01041=0.0000,5417.0162
EC01042=0.0000,5419.2050
EC01043=0.0000,5421.4028
EC01044=0.0000,5423.5971
EC01045=0.0000,5425.7952
EC01046=0.0000,5427.9837
EC01047=0.0000,5429.9842
EC01048=0.0000,5431.5162
EC01049=0.0000,5432.3970
EC01050=0.0000,5433.0583
EC01051=0.0000,5433.7518
EC01052=0.0000,5434.7152
EC01053=0.0000,5436.3389
EC01054=0.0000,5439.0399
EC01055=0.0000,5441.9437
EC01056=0.0000,5445.0000
EC01057=0.0000,5448.0563
EC01058=0.0000,5450.9601
EC01059=0.0000,5453.6611
EC01060=0.0000,5455.2848
EC01061=0.0000,5456.2482
EC01062=0.0000,5456.9417
EC01063=0.0000,5457.6030
EC01064=0.0000,5458.4838
EC01065=0.0000,5460.0158
EC01066=0.0000,5462.0163
EC01067=0.0000,5464.2048
EC01068=0.0000,5466.4029
EC01069=0.0000,5468.5972
EC01070=0.0000,5470.7950
EC01071=0.0000,5472.9838
EC01072=0.0000,5474.9845
EC01073=0.0000,5476.5163
EC01074=0.0000,5477.3970
EC01075=0.0000,5478.0583
EC01076=0.0000,5478.7517
EC01077=0.0000,5479.7148
EC01078=0.0000,5481.3390
EC01079=0.0000,5484.0402
EC01080=0.0000,5486.9435
EC01081=0.0000,5490.0000
EC01082=0.0000,5493.0565
EC01083=0.0000,5495.9604
EC01084=0.0000,5498.6610
EC01085=0.0000,5500.2852
EC01086=0.0000,5501.2483
EC01087=0.0000,5501.9417
EC01088=0.0000,5502.6030
EC01089=0.0000,5503.4837
EC01090=0.0000,5505.0155
EC01091=0.0000,5507.0162
EC01092=0.0000,5509.2050
EC01093=0.0000,5511.4028
EC01094=0.0000,5513.5971
EC01095=0.0000,5515.7952
EC01096=0.0000,5517.9837
EC01097=0.0000,5519.9842
EC01098=0.0000,5521.5162
EC01099=0.0000,5522.3970
EC01100=0.0000,5523.0583
EC01101=0.0000,5523.7518
EC01102=0.0000,5524.7152
EC01103=0.0000,5526.3389
EC01104=0.0000,5529.0399
EC01105=0.0000,5531.9437
EC01106=0.0000,5535.0000
EC01107=0.0000,5538.0563
EC01108=0.0000,5540.9601
EC01109=0.0000,5543.6611
EC01110=0.0000,5545.2848
EC01111=0.0000,5546.2482
EC01112=0.0000,5546.9417
EC01113=0.0000,5547.6030
EC01114=0.0000,5548.4838
EC01115=0.0000,5550.0158
EC01116=0.0000,5552.0163
EC01117=0.0000,5554.2048
EC01118=0.0000,5556.4029
EC01119=0.0000,5558.5972
EC01120=0.0000,5560.7950
EC01121=0.0000,5562.9838
EC01122=0.0000,5564.9845
EC01123=0.0000,5566.5163
EC01124=0.0000,5567.3970
EC01125=0.0000,5568.0583
EC01126=0.0000,5568.7517
EC01127=0.0000,5569.7148
EC01128=0.0000,5571.3390
EC01129=0.0000,5574.0402
EC01130=0.0000,5576.9435
EC01131=0.0000,5580.0000
EC01132=0.0000,5580.0000
EC01133=0.0000,5583.0565
EC01134=0.0000,5585.9604
EC01135=0.0000,5588.6610
EC01136=0.0000,5590.2852
EC01137=0.0000,5591.2483
EC01138=0.0000,5591.9417
EC01139=0.0000,5592.6030
EC01140=0.0000,5593.4837
EC01141=0.0000,5595.0155
EC01142=0.0000,5597.0162
EC01143=0.0000,5599.2050
EC01144=0.0000,5601.4028
EC01145=0.0000,5603.5971
EC01146=0.0000,5605.7952
EC01147=0.0000,5607.9837
EC01148=0.0000,5609.9842
EC01149=0.0000,5611.5162
EC01150=0.0000,5612.3970
EC01151=0.0000,5613.0583
EC01152=0.0000,5613.7518
EC01153=0.0000,5614.7152
EC01154=0.0000,5616.3389
EC01155=0.0000,5619.0399
EC01156=0.0000,5621.9437
EC01157=0.0000,5625.0000
EC01158=0.0000,5628.0563
EC01159=0.0000,5630.9601
EC01160=0.0000,5633.6611
EC01161=0.0000,5635.2848
EC01162=0.0000,5636.2482
EC01163=0.0000,5636.9417
EC01164=0.0000,5637.6030
EC01165=0.0000,5638.4838
EC01166=0.0000,5640.0158
EC01167=0.0000,5642.0163
EC01168=0.0000,5644.2048
EC01169=0.0000,5646.4029
EC01170=0.0000,5648.5972
EC01171=0.0000,5650.7950
EC01172=0.0000,5652.9838
EC01173=0.0000,5654.9845
EC01174=0.0000,5656.5163
EC01175=0.0000,5657.3970
EC01176=0.0000,5658.0583
EC01177=0.0000,5658.7517
EC01178=0.0000,5659.7148
EC01179=0.0000,5661.3390
EC01180=0.0000,5664.0402
EC01181=0.0000,5666.9435
EC01182=0.0000,5670.0000
EC01183=0.0000,5673.0565
EC01184=0.0000,5675.9604
EC01185=0.0000,5678.6610
EC01186=0.0000,5680.2852
EC01187=0.0000,5681.2483
EC01188=0.0000,5681.9417
EC01189=0.0000,5682.6030
EC01190=0.0000,5683.4837
EC01191=0.0000,5685.0155
EC01192=0.0000,5687.0162
EC01193=0.0000,5689.2050
EC01194=0.0000,5691.4028
EC01195=0.0000,5693.5971
EC01196=0.0000,5695.7952
EC01197=0.0000,5697.9837
EC01198=0.0000,5699.9842
EC01199=0.0000,5701.5162
EC01200=0.0000,5702.3970
EC01201=0.0000,5703.0583
EC01202=0.0000,5703.7518
EC01203=0.0000,5704.7152
EC01204=0.0000,5706.3389
EC01205=0.0000,5709.0399
EC01206=0.0000,5711.9437
EC01207=0.0000,5715.0000
EC01208=0.0000,5718.0563
EC01209=0.0000,5720.9601
EC01210=0.0000,5723.6611
EC01211=0.0000,5725.2848
EC01212=0.0000,5726.2482
EC01213=0.0000,5726.9417
EC01214=0.0000,5727.6030
EC01215=0.0000,5728.4838
EC01216=0.0000,5730.0158
EC01217=0.0000,5732.0163
EC01218=0.0000,5734.2048
EC01219=0.0000,5736.4029
EC01220=0.0000,5738.5972
EC01221=0.0000,5740.7950
EC01222=0.0000,5742.9838
EC01223=0.0000,5744.9845
EC01224=0.0000,5746.5163
EC01225=0.0000,5747.3970
EC01226=0.0000,5748.0583
EC01227=0.0000,5748.7517
EC01228=0.0000,5749.7148
EC01229=0.0000,5751.3390
EC01230=0.0000,5754.0396
EC01231=0.0000,5756.9435
EC01232=0.0000,5760.0000
EC01233=0.0000,5760.0000
EC01234=0.0000,5763.0242
EC01235=0.0000,5765.9175
EC01236=0.0000,5768.6252
EC01237=0.0000,5770.2250
EC01238=0.0000,5771.1519
EC01239=0.0000,5771.8065
EC01240=0.0000,5772.4248
EC01241=0.0000,5773.2580
EC01242=0.0000,5774.7847
EC01243=0.0000,5776.8204
EC01244=0.0000,5779.0758
EC01245=0.0000,5781.3580
EC01246=0.0000,5783.6417
EC01247=0.0000,5785.9241
EC01248=0.0000,5788.1796
EC01249=0.0000,5790.2155
EC01250=0.0000,5791.7418
EC01251=0.0000,5792.5751
EC01252=0.0000,5793.1936
EC01253=0.0000,5793.8475
EC01254=0.0000,5794.7753
EC01255=0.0000,5796.3747
EC01256=0.0000,5799.0826
EC01257=0.0000,5801.9754
EC01258=0.0000,5805.0000
EC01259=0.0000,5808.0237
EC01260=0.0000,5810.9174
EC01261=0.0000,5813.6253
EC01262=0.0000,5815.2247
EC01263=0.0000,5816.1525
EC01264=0.0000,5816.8064
EC01265=0.0000,5817.4249
EC01266=0.0000,5818.2582
EC01267=0.0000,5819.7845
EC01268=0.0000,5821.8204
EC01269=0.0000,5824.0759
EC01270=0.0000,5826.3583
EC01271=0.0000,5828.6420
EC01272=0.0000,5830.9242
EC01273=0.0000,5833.1796
EC01274=0.0000,5835.2153
EC01275=0.0000,5836.7420
EC01276=0.0000,5837.5752
EC01277=0.0000,5838.1935
EC01278=0.0000,5838.8481
EC01279=0.0000,5839.7750
EC01280=0.0000,5841.3748
EC01281=0.0000,5844.0825
EC01282=0.0000,5846.9758
EC01283=0.0000,5850.0000
EC01284=0.0000,5853.0242
EC01285=0.0000,5855.9175
EC01286=0.0000,5858.6252
EC01287=0.0000,5860.2250
EC01288=0.0000,5861.1519
EC01289=0.0000,5861.8065
EC01290=0.0000,5862.4248
EC01291=0.0000,5863.2580
EC01292=0.0000,5864.7847
EC01293=0.0000,5866.8204
EC01294=0.0000,5869.0758
EC01295=0.0000,5871.3580
EC01296=0.0000,5873.6417
EC01297=0.0000,5875.9241
EC01298=0.0000,5878.1796
EC01299=0.0000,5880.2155
EC01300=0.0000,5881.7418
EC01301=0.0000,5882.5751
EC01302=0.0000,5883.1936
EC01303=0.0000,5883.8475
EC01304=0.0000,5884.7753
EC01305=0.0000,5886.3747
EC01306=0.0000,5889.0826
EC01307=0.0000,5891.9754
EC01308=0.0000,5895.0000
EC01309=0.0000,5898.0237
EC01310=0.0000,5900.9174
EC01311=0.0000,5903.6253
EC01312=0.0000,5905.2247
EC01313=0.0000,5906.1525
EC01314=0.0000,5906.8064
EC01315=0.0000,5907.4249
EC01316=0.0000,5908.2582
EC01317=0.0000,5909.7845
EC01318=0.0000,5911.8204
EC01319=0.0000,5914.0759
EC01320=0.0000,5916.3583
EC01321=0.0000,5918.6420
EC01322=0.0000,5920.9242
EC01323=0.0000,5923.1796
EC01324=0.0000,5925.2153
EC01325=0.0000,5926.7420
EC01326=0.0000,5927.5752
EC01327=0.0000,5928.1935
EC01328=0.0000,5928.8481
EC01329=0.0000,5929.7750
EC01330=0.0000,5931.3748
EC01331=0.0000,5934.0825
EC01332=0.0000,5936.9758
EC01333=0.0000,5940.0000
EC01334=0.0000,5940.0000
EC01335=0.0000,5943.0242
EC01336=0.0000,5945.9175
EC01337=0.0000,5948.6252
EC01338=0.0000,5950.2250
EC01339=0.0000,5951.1519
EC01340=0.0000,5951.8065
EC01341=0.0000,5952.4248
EC01342=0.0000,5953.2580
EC01343=0.0000,5954.7847
EC01344=0.0000,5956.8204
EC01345=0.0000,5959.0758
EC01346=0.0000,5961.3580
EC01347=0.0000,5963.6417
EC01348=0.0000,5965.9241
EC01349=0.0000,5968.1796
EC01350=0.0000,5970.2155
EC01351=0.0000,5971.7418
EC01352=0.0000,5972.5751
EC01353=0.0000,5973.1936
EC01354=0.0000,5973.8475
EC01355=0.0000,5974.7753
EC01356=0.0000,5976.3747
EC01357=0.0000,5979.0826
EC01358=0.0000,5981.9754
EC01359=0.0000,5985.0000
EC01360=0.0000,5988.0237
EC01361=0.0000,5990.9174
EC01362=0.0000,5993.6253
EC01363=0.0000,5995.2247
EC01364=0.0000,5996.1525
EC01365=0.0000,5996.8064
EC01366=0.0000,5997.4249
EC01367=0.0000,5998.2582
EC01368=0.0000,5999.7845
EC01369=0.0000,6001.8204
EC01370=0.0000,6004.0759
EC01371=0.0000,6006.3583
EC01372=0.0000,6008.6420
EC01373=0.0000,6010.9242
EC01374=0.0000,6013.1796
EC01375=0.0000,6015.2153
EC01376=0.0000,6016.7420
EC01377=0.0000,6017.5752
EC01378=0.0000,6018.1935
EC01379=0.0000,6018.8481
EC01380=0.0000,6019.7750
EC01381=0.0000,6021.3748
EC01382=0.0000,6024.0825
EC01383=0.0000,6026.9758
EC01384=0.0000,6030.0000
EC01385=0.0000,6033.0242
EC01386=0.0000,6035.9175
EC01387=0.0000,6038.6252
EC01388=0.0000,6040.2250
EC01389=0.0000,6041.1519
EC01390=0.0000,6041.8065
EC01391=0.0000,6042.4248
EC01392=0.0000,6043.2580
EC01393=0.0000,6044.7847
EC01394=0.0000,6046.8204
EC01395=0.0000,6049.0758
EC01396=0.0000,6051.3580
EC01397=0.0000,6053.6417
EC01398=0.0000,6055.9241
EC01399=0.0000,6058.1796
EC01400=0.0000,6060.2155
EC01401=0.0000,6061.7418
EC01402=0.0000,6062.5751
EC01403=0.0000,6063.1936
EC01404=0.0000,6063.8475
EC01405=0.0000,6064.7753
EC01406=0.0000,6066.3747
EC01407=0.0000,6069.0826
EC01408=0.0000,6071.9754
EC01409=0.0000,6075.0000
EC01410=0.0000,6078.0237
EC01411=0.0000,6080.9174
EC01412=0.0000,6083.6253
EC01413=0.0000,6085.2247
EC01414=0.0000,6086.1525
EC01415=0.0000,6086.8064
EC01416=0.0000,6087.4249
EC01417=0.0000,6088.2582
EC01418=0.0000,6089.7845
EC01419=0.0000,6091.8204
EC01420=0.0000,6094.0759
EC01421=0.0000,6096.3583
EC01422=0.0000,6098.6420
EC01423=0.0000,6100.9242
EC01424=0.0000,6103.1796
EC01425=0.0000,6105.2153
EC01426=0.0000,6106.7420
EC01427=0.0000,6107.5752
EC01428=0.0000,6108.1935
EC01429=0.0000,6108.8481
EC01430=0.0000,6109.7750
EC01431=0.0000,6111.3748
EC01432=0.0000,6114.0825
EC01433=0.0000,6116.9758
EC01434=0.0000,6120.0000
EC01435=0.0000,6120.0000
EC01436=0.0000,6122.9903
EC01437=0.0000,6125.8729
EC01438=0.0000,6128.5881
EC01439=0.0000,6130.1621
EC01440=0.0000,6131.0515
EC01441=0.0000,6131.6656
EC01442=0.0000,6132.2395
EC01443=0.0000,6133.0258
EC01444=0.0000,6134.5467
EC01445=0.0000,6136.6187
EC01446=0.0000,6138.9437
EC01447=0.0000,6141.3119
EC01448=0.0000,6143.6874
EC01449=0.0000,6146.0569
EC01450=0.0000,6148.3812
EC01451=0.0000,6150.4534
EC01452=0.0000,6151.9748
EC01453=0.0000,6152.7607
EC01454=0.0000,6153.3343
EC01455=0.0000,6153.9482
EC01456=0.0000,6154.8381
EC01457=0.0000,6156.4120
EC01458=0.0000,6159.1268
EC01459=0.0000,6162.0095
EC01460=0.0000,6165.0000
EC01461=0.0000,6167.9905
EC01462=0.0000,6170.8732
EC01463=0.0000,6173.5880
EC01464=0.0000,6175.1619
EC01465=0.0000,6176.0518
EC01466=0.0000,6176.6657
EC01467=0.0000,6177.2393
EC01468=0.0000,6178.0252
EC01469=0.0000,6179.5466
EC01470=0.0000,6181.6188
EC01471=0.0000,6183.9431
EC01472=0.0000,6186.3126
EC01473=0.0000,6188.6881
EC01474=0.0000,6191.0563
EC01475=0.0000,6193.3813
EC01476=0.0000,6195.4533
EC01477=0.0000,6196.9742
EC01478=0.0000,6197.7605
EC01479=0.0000,6198.3344
EC01480=0.0000,6198.9485
EC01481=0.0000,6199.8379
EC01482=0.0000,6201.4119
EC01483=0.0000,6204.1271
EC01484=0.0000,6207.0097
EC01485=0.0000,6210.0000
EC01486=0.0000,6212.9903
EC01487=0.0000,6215.8729
EC01488=0.0000,6218.5881
EC01489=0.0000,6220.1621
EC01490=0.0000,6221.0515
EC01491=0.0000,6221.6656
EC01492=0.0000,6222.2395
EC01493=0.0000,6223.0258
EC01494=0.0000,6224.5467
EC01495=0.0000,6226.6187
EC01496=0.0000,6228.9437
EC01497=0.0000,6231.3119
EC01498=0.0000,6233.6874
EC01499=0.0000,6236.0569
EC01500=0.0000,6238.3812
EC01501=0.0000,6240.4534
EC01502=0.0000,6241.9748
EC01503=0.0000,6242.7607
EC01504=0.0000,6243.3343
EC01505=0.0000,6243.9482
EC01506=0.0000,6244.8381
EC01507=0.0000,6246.4120
EC01508=0.0000,6249.1268
EC01509=0.0000,6252.0095
EC01510=0.0000,6255.0000
EC01511=0.0000,6257.9905
EC01512=0.0000,6260.8732
EC01513=0.0000,6263.5880
EC01514=0.0000,6265.1619
EC01515=0.0000,6266.0518
EC01516=0.0000,6266.6657
EC01517=0.0000,6267.2393
EC01518=0.0000,6268.0252
EC01519=0.0000,6269.5466
EC01520=0.0000,6271.6188
EC01521=0.0000,6273.9431
EC01522=0.0000,6276.3126
EC01523=0.0000,6278.6881
EC01524=0.0000,6281.0563
EC01525=0.0000,6283.3813
EC01526=0.0000,6285.4533
EC01527=0.0000,6286.9742
EC01528=0.0000,6287.7605
EC01529=0.0000,6288.3344
EC01530=0.0000,6288.9485
EC01531=0.0000,6289.8379
EC01532=0.0000,6291.4119
EC01533=0.0000,6294.1271
EC01534=0.0000,6297.0097
EC01535=0.0000,6300.0000
EC01536=0.0000,6300.0000
EC01537=0.0000,6302.9903
EC01538=0.0000,6305.8729
EC01539=0.0000,6308.5881
EC01540=0.0000,6310.1621
EC01541=0.0000,6311.0515
EC01542=0.0000,6311.6656
EC01543=0.0000,6312.2395
EC01544=0.0000,6313.0258
EC01545=0.0000,6314.5467
EC01546=0.0000,6316.6187
EC01547=0.0000,6318.9437
EC01548=0.0000,6321.3119
EC01549=0.0000,6323.6874
EC01550=0.0000,6326.0569
EC01551=0.0000,6328.3812
EC01552=0.0000,6330.4534
EC01553=0.0000,6331.9748
EC01554=0.0000,6332.7607
EC01555=0.0000,6333.3343
EC01556=0.0000,6333.9482
EC01557=0.0000,6334.8381
EC01558=0.0000,6336.4120
EC01559=0.0000,6339.1268
EC01560=0.0000,6342.0095
EC01561=0.0000,6345.0000
EC01562=0.0000,6347.9905
EC01563=0.0000,6350.8732
EC01564=0.0000,6353.5880
EC01565=0.0000,6355.1619
EC01566=0.0000,6356.0518
EC01567=0.0000,6356.6657
EC01568=0.0000,6357.2393
EC01569=0.0000,6358.0252
EC01570=0.0000,6359.5466
EC01571=0.0000,6361.6188
EC01572=0.0000,6363.9431
EC01573=0.0000,6366.3126
EC01574=0.0000,6368.6881
EC01575=0.0000,6371.0563
EC01576=0.0000,6373.3813
EC01577=0.0000,6375.4533
EC01578=0.0000,6376.9742
EC01579=0.0000,6377.7605
EC01580=0.0000,6378.3344
EC01581=0.0000,6378.9485
EC01582=0.0000,6379.8379
EC01583=0.0000,6381.4119
EC01584=0.0000,6384.1271
EC01585=0.0000,6387.0097
EC01586=0.0000,6390.0000
EC01587=0.0000,6392.9903
EC01588=0.0000,6395.8729
EC01589=0.0000,6398.5881
EC01590=0.0000,6400.1621
EC01591=0.0000,6401.0515
EC01592=0.0000,6401.6656
EC01593=0.0000,6402.2395
EC01594=0.0000,6403.0258
EC01595=0.0000,6404.5467
EC01596=0.0000,6406.6187
EC01597=0.0000,6408.9437
EC01598=0.0000,6411.3119
EC01599=0.0000,6413.6874
EC01600=0.0000,6416.0569
EC01601=0.0000,6418.3812
EC01602=0.0000,6420.4534
EC01603=0.0000,6421.9748
EC01604=0.0000,6422.7607
EC01605=0.0000,6423.3343
EC01606=0.0000,6423.9482
EC01607=0.0000,6424.8381
EC01608=0.0000,6426.4120
EC01609=0.0000,6429.1268
EC01610=0.0000,6432.0095
EC01611=0.0000,6435.0000
EC01612=0.0000,6437.9905
EC01613=0.0000,6440.8732
EC01614=0.0000,6443.5880
EC01615=0.0000,6445.1619
EC01616=0.0000,6446.0518
EC01617=0.0000,6446.6657
EC01618=0.0000,6447.2393
EC01619=0.0000,6448.0252
EC01620=0.0000,6449.5466
EC01621=0.0000,6451.6188
EC01622=0.0000,6453.9431
EC01623=0.0000,6456.3126
EC01624=0.0000,6458.6881
EC01625=0.0000,6461.0563
EC01626=0.0000,6463.3813
EC01627=0.0000,6465.4533
EC01628=0.0000,6466.9742
EC01629=0.0000,6467.7605
EC01630=0.0000,6468.3344
EC01631=0.0000,6468.9485
EC01632=0.0000,6469.8379
EC01633=0.0000,6471.4119
EC01634=0.0000,6474.1271
EC01635=0.0000,6477.0097
EC01636=0.0000,6480.0000
EC01637=0.0000,6480.0000
EC01638=0.0000,6482.9548
EC01639=0.0000,6485.8263
EC01640=0.0000,6488.5486
EC01641=0.0000,6490.0964
EC01642=0.0000,6490.9471
EC01643=0.0000,6491.5198
EC01644=0.0000,6492.0484
EC01645=0.0000,6492.7860
EC01646=0.0000,6494.3034
EC01647=0.0000,6496.4132
EC01648=0.0000,6498.8079
EC01649=0.0000,6501.2653
EC01650=0.0000,6503.7346
EC01651=0.0000,6506.1917
EC01652=0.0000,6508.5867
EC01653=0.0000,6510.6966
EC01654=0.0000,6512.2136
EC01655=0.0000,6512.9519
EC01656=0.0000,6513.4806
EC01657=0.0000,6514.0527
EC01658=0.0000,6514.9034
EC01659=0.0000,6516.4513
EC01660=0.0000,6519.1737
EC01661=0.0000,6522.0450
EC01662=0.0000,6525.0000
EC01663=0.0000,6527.9550
EC01664=0.0000,6530.8263
EC01665=0.0000,6533.5487
EC01666=0.0000,6535.0966
EC01667=0.0000,6535.9473
EC01668=0.0000,6536.5194
EC01669=0.0000,6537.0481
EC01670=0.0000,6537.7864
EC01671=0.0000,6539.3034
EC01672=0.0000,6541.4133
EC01673=0.0000,6543.8083
EC01674=0.0000,6546.2654
EC01675=0.0000,6548.7347
EC01676=0.0000,6551.1921
EC01677=0.0000,6553.5868
EC01678=0.0000,6555.6966
EC01679=0.0000,6557.2140
EC01680=0.0000,6557.9516
EC01681=0.0000,6558.4802
EC01682=0.0000,6559.0529
EC01683=0.0000,6559.9036
EC01684=0.0000,6561.4514
EC01685=0.0000,6564.1737
EC01686=0.0000,6567.0452
EC01687=0.0000,6570.0000
EC01688=0.0000,6572.9548
EC01689=0.0000,6575.8263
EC01690=0.0000,6578.5486
EC01691=0.0000,6580.0964
EC01692=0.0000,6580.9471
EC01693=0.0000,6581.5198
EC01694=0.0000,6582.0484
EC01695=0.0000,6582.7860
EC01696=0.0000,6584.3034
EC01697=0.0000,6586.4132
EC01698=0.0000,6588.8079
EC01699=0.0000,6591.2653
EC01700=0.0000,6593.7346
EC01701=0.0000,6596.1917
EC01702=0.0000,6598.5867
EC01703=0.0000,6600.6966
EC01704=0.0000,6602.2136
EC01705=0.0000,6602.9519
EC01706=0.0000,6603.4806
EC01707=0.0000,6604.0527
EC01708=0.0000,6604.9034
EC01709=0.0000,6606.4513
EC01710=0.0000,6609.1737
EC01711=0.0000,6612.0450
EC01712=0.0000,6615.0000
EC01713=0.0000,6617.9550
EC01714=0.0000,6620.8263
EC01715=0.0000,6623.5487
EC01716=0.0000,6625.0966
EC01717=0.0000,6625.9473
EC01718=0.0000,6626.5194
EC01719=0.0000,6627.0481
EC01720=0.0000,6627.7864
EC01721=0.0000,6629.3034
EC01722=0.0000,6631.4133
EC01723=0.0000,6633.8083
EC01724=0.0000,6636.2654
EC01725=0.0000,6638.7347
EC01726=0.0000,6641.1921
EC01727=0.0000,6643.5868
EC01728=0.0000,6645.6966
EC01729=0.0000,6647.2140
EC01730=0.0000,6647.9516
EC01731=0.0000,6648.4802
EC01732=0.0000,6649.0529
EC01733=0.0000,6649.9036
EC01734=0.0000,6651.4514
EC01735=0.0000,6654.1737
EC01736=0.0000,6657.0452
EC01737=0.0000,6660.0000
EC01738=0.0000,6660.0000
EC01739=0.0000,6662.9548
EC01740=0.0000,6665.8263
EC01741=0.0000,6668.5486
EC01742=0.0000,6670.0964
EC01743=0.0000,6670.9471
EC01744=0.0000,6671.5198
EC01745=0.0000,6672.0484
EC01746=0.0000,6672.7860
EC01747=0.0000,6674.3034
EC01748=0.0000,6676.4132
EC01749=0.0000,6678.8079
EC01750=0.0000,6681.2653
EC01751=0.0000,6683.7346
EC01752=0.0000,6686.1917
EC01753=0.0000,6688.5867
EC01754=0.0000,6690.6966
EC01755=0.0000,6692.2136
EC01756=0.0000,6692.9519
EC01757=0.0000,6693.4806
EC01758=0.0000,6694.0527
EC01759=0.0000,6694.9034
EC01760=0.0000,6696.4513
EC01761=0.0000,6699.1737
EC01762=0.0000,6702.0450
EC01763=0.0000,6705.0000
EC01764=0.0000,6707.9550
EC01765=0.0000,6710.8263
EC01766=0.0000,6713.5487
EC01767=0.0000,6715.0966
EC01768=0.0000,6715.9473
EC01769=0.0000,6716.5194
EC01770=0.0000,6717.0481
EC01771=0.0000,6717.7864
EC01772=0.0000,6719.3034
EC01773=0.0000,6721.4133
EC01774=0.0000,6723.8083
EC01775=0.0000,6726.2654
EC01776=0.0000,6728.7347
EC01777=0.0000,6731.1921
EC01778=0.0000,6733.5868
EC01779=0.0000,6735.6966
EC01780=0.0000,6737.2140
EC01781=0.0000,6737.9516
EC01782=0.0000,6738.4802
EC01783=0.0000,6739.0529
EC01784=0.0000,6739.9036
EC01785=0.0000,6741.4514
EC01786=0.0000,6744.1737
EC01787=0.0000,6747.0452
EC01788=0.0000,6750.0000
EC01789=0.0000,6752.9548
EC01790=0.0000,6755.8263
EC01791=0.0000,6758.5486
EC01792=0.0000,6760.0964
EC01793=0.0000,6760.9471
EC01794=0.0000,6761.5198
EC01795=0.0000,6762.0484
EC01796=0.0000,6762.7860
EC01797=0.0000,6764.3034
EC01798=0.0000,6766.4132
EC01799=0.0000,6768.8079
EC01800=0.0000,6771.2653
EC01801=0.0000,6773.7346
EC01802=0.0000,6776.1917
EC01803=0.0000,6778.5867
EC01804=0.0000,6780.6966
EC01805=0.0000,6782.2136
EC01806=0.0000,6782.9519
EC01807=0.0000,6783.4806
EC01808=0.0000,6784.0527
EC01809=0.0000,6784.9034
EC01810=0.0000,6786.4513
EC01811=0.0000,6789.1737
EC01812=0.0000,6792.0450
EC01813=0.0000,6795.0000
EC01814=0.0000,6797.9550
EC01815=0.0000,6800.8263
EC01816=0.0000,6803.5487
EC01817=0.0000,6805.0966
EC01818=0.0000,6805.9473
EC01819=0.0000,6806.5194
EC01820=0.0000,6807.0481
EC01821=0.0000,6807.7864
EC01822=0.0000,6809.3034
EC01823=0.0000,6811.4133
EC01824=0.0000,6813.8083
EC01825=0.0000,6816.2654
EC01826=0.0000,6818.7347
EC01827=0.0000,6821.1921
EC01828=0.0000,6823.5868
EC01829=0.0000,6825.6966
EC01830=0.0000,6827.2140
EC01831=0.0000,6827.9516
EC01832=0.0000,6828.4802
EC01833=0.0000,6829.0529
EC01834=0.0000,6829.9036
EC01835=0.0000,6831.4514
EC01836=0.0000,6834.1737
EC01837=0.0000,6837.0452
EC01838=0.0000,6840.0000
EC01839=0.0000,6840.0000
EC01840=0.0000,6842.9180
EC01841=0.0000,6845.7775
EC01842=0.0000,6848.5076
EC01843=0.0000,6850.0280
EC01844=0.0000,6850.8382
EC01845=0.0000,6851.3683
EC01846=0.0000,6851.8512
EC01847=0.0000,6852.5410
EC01848=0.0000,6854.0550
EC01849=0.0000,6856.2037
EC01850=0.0000,6858.6701
EC01851=0.0000,6861.2180
EC01852=0.0000,6863.7821
EC01853=0.0000,6866.3297
EC01854=0.0000,6868.7961
EC01855=0.0000,6870.9450
EC01856=0.0000,6872.4587
EC01857=0.0000,6873.1487
EC01858=0.0000,6873.6320
EC01859=0.0000,6874.1614
EC01860=0.0000,6874.9722
EC01861=0.0000,6876.4919
EC01862=0.0000,6879.2230
EC01863=0.0000,6882.0820
EC01864=0.0000,6885.0000
EC01865=0.0000,6887.9180
EC01866=0.0000,6890.7770
EC01867=0.0000,6893.5081
EC01868=0.0000,6895.0278
EC01869=0.0000,6895.8386
EC01870=0.0000,6896.3680
EC01871=0.0000,6896.8513
EC01872=0.0000,6897.5413
EC01873=0.0000,6899.0550
EC01874=0.0000,6901.2039
EC01875=0.0000,6903.6703
EC01876=0.0000,6906.2179
EC01877=0.0000,6908.7820
EC01878=0.0000,6911.3299
EC01879=0.0000,6913.7963
EC01880=0.0000,6915.9450
EC01881=0.0000,6917.4590
EC01882=0.0000,6918.1488
EC01883=0.0000,6918.6317
EC01884=0.0000,6919.1618
EC01885=0.0000,6919.9720
EC01886=0.0000,6921.4924
EC01887=0.0000,6924.2225
EC01888=0.0000,6927.0820
EC01889=0.0000,6930.0000
EC01890=0.0000,6932.9180
EC01891=0.0000,6935.7775
EC01892=0.0000,6938.5076
EC01893=0.0000,6940.0280
EC01894=0.0000,6940.8382
EC01895=0.0000,6941.3683
EC01896=0.0000,6941.8512
EC01897=0.0000,6942.5410
EC01898=0.0000,6944.0550
EC01899=0.0000,6946.2037
EC01900=0.0000,6948.6701
EC01901=0.0000,6951.2180
EC01902=0.0000,6953.7821
EC01903=0.0000,6956.3297
EC01904=0.0000,6958.7961
EC01905=0.0000,6960.9450
EC01906=0.0000,6962.4587
EC01907=0.0000,6963.1487
EC01908=0.0000,6963.6320
EC01909=0.0000,6964.1614
EC01910=0.0000,6964.9722
EC01911=0.0000,6966.4919
EC01912=0.0000,6969.2230
EC01913=0.0000,6972.0820
EC01914=0.0000,6975.0000
EC01915=0.0000,6977.9180
EC01916=0.0000,6980.7770
EC01917=0.0000,6983.5081
EC01918=0.0000,6985.0278
EC01919=0.0000,6985.8386
EC01920=0.0000,6986.3680
EC01921=0.0000,6986.8513
EC01922=0.0000,6987.5413
EC01923=0.0000,6989.0550
EC01924=0.0000,6991.2039
EC01925=0.0000,6993.6703
EC01926=0.0000,6996.2179
EC01927=0.0000,6998.7820
EC01928=0.0000,7001.3299
EC01929=0.0000,7003.7963
EC01930=0.0000,7005.9450
EC01931=0.0000,7007.4590
EC01932=0.0000,7008.1488
EC01933=0.0000,7008.6317
EC01934=0.0000,7009.1618
EC01935=0.0000,7009.9720
EC01936=0.0000,7011.4924
EC01937=0.0000,7014.2225
EC01938=0.0000,7017.0820
EC01939=0.0000,7020.0000
EC01940=0.0000,7020.0000
EC01941=0.0000,7022.9180
EC01942=0.0000,7025.7775
EC01943=0.0000,7028.5076
EC01944=0.0000,7030.0280
EC01945=0.0000,7030.8382
EC01946=0.0000,7031.3683
EC01947=0.0000,7031.8512
EC01948=0.0000,7032.5410
EC01949=0.0000,7034.0550
EC01950=0.0000,7036.2037
EC01951=0.0000,7038.6701
EC01952=0.0000,7041.2180
EC01953=0.0000,7043.7821
EC01954=0.0000,7046.3297
EC01955=0.0000,7048.7961
EC01956=0.0000,7050.9450
EC01957=0.0000,7052.4587
EC01958=0.0000,7053.1487
EC01959=0.0000,7053.6320
EC01960=0.0000,7054.1614
EC01961=0.0000,7054.9722
EC01962=0.0000,7056.4919
EC01963=0.0000,7059.2230
EC01964=0.0000,7062.0820
EC01965=0.0000,7065.0000
EC01966=0.0000,7067.9180
EC01967=0.0000,7070.7770
EC01968=0.0000,7073.5081
EC01969=0.0000,7075.0278
EC01970=0.0000,7075.8386
EC01971=0.0000,7076.3680
EC01972=0.0000,7076.8513
EC01973=0.0000,7077.5413
EC01974=0.0000,7079.0550
EC01975=0.0000,7081.2039
EC01976=0.0000,7083.6703
EC01977=0.0000,7086.2179
EC01978=0.0000,7088.7820
EC01979=0.0000,7091.3299
EC01980=0.0000,7093.7963
EC01981=0.0000,7095.9450
EC01982=0.0000,7097.4590
EC01983=0.0000,7098.1488
EC01984=0.0000,7098.6317
EC01985=0.0000,7099.1618
EC01986=0.0000,7099.9720
EC01987=0.0000,7101.4924
EC01988=0.0000,7104.2225
EC01989=0.0000,7107.0820
EC01990=0.0000,7110.0000
EC01991=0.0000,7112.9180
EC01992=0.0000,7115.7775
EC01993=0.0000,7118.5076
EC01994=0.0000,7120.0280
EC01995=0.0000,7120.8382
EC01996=0.0000,7121.3683
EC01997=0.0000,7121.8512
EC01998=0.0000,7122.5410
EC01999=0.0000,7124.0550
//INST
///DATE 2021/02/10 13:51
///COMM
///ATTR SC,RW,RJ
////FRAME USER 2
///GROUP1 RB1
///GROUP2 ST1
NOP
SMOVL C00000 +MOVJ EC00000
SMOVL C00001 +MOVJ EC00001
SMOVL C00002 +MOVJ EC00002
SMOVL C00003 +MOVJ EC00003
SMOVL C00004 +MOVJ EC00004
SMOVL C00005 +MOVJ EC00005
SMOVL C00006 +MOVJ EC00006
SMOVL C00007 +MOVJ EC00007
SMOVL C00008 +MOVJ EC00008
SMOVL C00009 +MOVJ EC00009
SMOVL C00010 +MOVJ EC00010
SMOVL C00011 +MOVJ EC00011
SMOVL C00012 +MOVJ EC00012
SMOVL C00013 +MOVJ EC00013
SMOVL C00014 +MOVJ EC00014
SMOVL C00015 +MOVJ EC00015
SMOVL C00016 +MOVJ EC00016
SMOVL C00017 +MOVJ EC00017
SMOVL C00018 +MOVJ EC00018
SMOVL C00019 +MOVJ EC00019
SMOVL C00020 +MOVJ EC00020
SMOVL C00021 +MOVJ EC00021
SMOVL C00022 +MOVJ EC00022
SMOVL C00023 +MOVJ EC00023
SMOVL C00024 +MOVJ EC00024
SMOVL C00025 +MOVJ EC00025
SMOVL C00026 +MOVJ EC00026
SMOVL C00027 +MOVJ EC00027
SMOVL C00028 +MOVJ EC00028
SMOVL C00029 +MOVJ EC00029
SMOVL C00030 +MOVJ EC00030
SMOVL C00031 +MOVJ EC00031
SMOVL C00032 +MOVJ EC00032
SMOVL C00033 +MOVJ EC00033
SMOVL C00034 +MOVJ EC00034
SMOVL C00035 +MOVJ EC00035
SMOVL C00036 +MOVJ EC00036
SMOVL C00037 +MOVJ EC00037
SMOVL C00038 +MOVJ EC00038
SMOVL C00039 +MOVJ EC00039
SMOVL C00040 +MOVJ EC00040
SMOVL C00041 +MOVJ EC00041
SMOVL C00042 +MOVJ EC00042
SMOVL C00043 +MOVJ EC00043
SMOVL C00044 +MOVJ EC00044
SMOVL C00045 +MOVJ EC00045
SMOVL C00046 +MOVJ EC00046
SMOVL C00047 +MOVJ EC00047
SMOVL C00048 +MOVJ EC00048
SMOVL C00049 +MOVJ EC00049
SMOVL C00050 +MOVJ EC00050
SMOVL C00051 +MOVJ EC00051
SMOVL C00052 +MOVJ EC00052
SMOVL C00053 +MOVJ EC00053
SMOVL C00054 +MOVJ EC00054
SMOVL C00055 +MOVJ EC00055
SMOVL C00056 +MOVJ EC00056
SMOVL C00057 +MOVJ EC00057
SMOVL C00058 +MOVJ EC00058
SMOVL C00059 +MOVJ EC00059
SMOVL C00060 +MOVJ EC00060
SMOVL C00061 +MOVJ EC00061
SMOVL C00062 +MOVJ EC00062
SMOVL C00063 +MOVJ EC00063
SMOVL C00064 +MOVJ EC00064
SMOVL C00065 +MOVJ EC00065
SMOVL C00066 +MOVJ EC00066
SMOVL C00067 +MOVJ EC00067
SMOVL C00068 +MOVJ EC00068
SMOVL C00069 +MOVJ EC00069
SMOVL C00070 +MOVJ EC00070
SMOVL C00071 +MOVJ EC00071
SMOVL C00072 +MOVJ EC00072
SMOVL C00073 +MOVJ EC00073
SMOVL C00074 +MOVJ EC00074
SMOVL C00075 +MOVJ EC00075
SMOVL C00076 +MOVJ EC00076
SMOVL C00077 +MOVJ EC00077
SMOVL C00078 +MOVJ EC00078
SMOVL C00079 +MOVJ EC00079
SMOVL C00080 +MOVJ EC00080
SMOVL C00081 +MOVJ EC00081
SMOVL C00082 +MOVJ EC00082
SMOVL C00083 +MOVJ EC00083
SMOVL C00084 +MOVJ EC00084
SMOVL C00085 +MOVJ EC00085
SMOVL C00086 +MOVJ EC00086
SMOVL C00087 +MOVJ EC00087
SMOVL C00088 +MOVJ EC00088
SMOVL C00089 +MOVJ EC00089
SMOVL C00090 +MOVJ EC00090
SMOVL C00091 +MOVJ EC00091
SMOVL C00092 +MOVJ EC00092
SMOVL C00093 +MOVJ EC00093
SMOVL C00094 +MOVJ EC00094
SMOVL C00095 +MOVJ EC00095
SMOVL C00096 +MOVJ EC00096
SMOVL C00097 +MOVJ EC00097
SMOVL C00098 +MOVJ EC00098
SMOVL C00099 +MOVJ EC00099
SMOVL C00100 +MOVJ EC00100
SMOVL C00101 +MOVJ EC00101
SMOVL C00102 +MOVJ EC00102
SMOVL C00103 +MOVJ EC00103
SMOVL C00104 +MOVJ EC00104
SMOVL C00105 +MOVJ EC00105
SMOVL C00106 +MOVJ EC00106
SMOVL C00107 +MOVJ EC00107
SMOVL C00108 +MOVJ EC00108
SMOVL C00109 +MOVJ EC00109
SMOVL C00110 +MOVJ EC00110
SMOVL C00111 +MOVJ EC00111
SMOVL C00112 +MOVJ EC00112
SMOVL C00113 +MOVJ EC00113
SMOVL C00114 +MOVJ EC00114
SMOVL C00115 +MOVJ EC00115
SMOVL C00116 +MOVJ EC00116
SMOVL C00117 +MOVJ EC00117
SMOVL C00118 +MOVJ EC00118
SMOVL C00119 +MOVJ EC00119
SMOVL C00120 +MOVJ EC00120
SMOVL C00121 +MOVJ EC00121
SMOVL C00122 +MOVJ EC00122
SMOVL C00123 +MOVJ EC00123
SMOVL C00124 +MOVJ EC00124
SMOVL C00125 +MOVJ EC00125
SMOVL C00126 +MOVJ EC00126
SMOVL C00127 +MOVJ EC00127
SMOVL C00128 +MOVJ EC00128
SMOVL C00129 +MOVJ EC00129
SMOVL C00130 +MOVJ EC00130
SMOVL C00131 +MOVJ EC00131
SMOVL C00132 +MOVJ EC00132
SMOVL C00133 +MOVJ EC00133
SMOVL C00134 +MOVJ EC00134
SMOVL C00135 +MOVJ EC00135
SMOVL C00136 +MOVJ EC00136
SMOVL C00137 +MOVJ EC00137
SMOVL C00138 +MOVJ EC00138
SMOVL C00139 +MOVJ EC00139
SMOVL C00140 +MOVJ EC00140
SMOVL C00141 +MOVJ EC00141
SMOVL C00142 +MOVJ EC00142
SMOVL C00143 +MOVJ EC00143
SMOVL C00144 +MOVJ EC00144
SMOVL C00145 +MOVJ EC00145
SMOVL C00146 +MOVJ EC00146
SMOVL C00147 +MOVJ EC00147
SMOVL C00148 +MOVJ EC00148
SMOVL C00149 +MOVJ EC00149
SMOVL C00150 +MOVJ EC00150
SMOVL C00151 +MOVJ EC00151
SMOVL C00152 +MOVJ EC00152
SMOVL C00153 +MOVJ EC00153
SMOVL C00154 +MOVJ EC00154
SMOVL C00155 +MOVJ EC00155
SMOVL C00156 +MOVJ EC00156
SMOVL C00157 +MOVJ EC00157
SMOVL C00158 +MOVJ EC00158
SMOVL C00159 +MOVJ EC00159
SMOVL C00160 +MOVJ EC00160
SMOVL C00161 +MOVJ EC00161
SMOVL C00162 +MOVJ EC00162
SMOVL C00163 +MOVJ EC00163
SMOVL C00164 +MOVJ EC00164
SMOVL C00165 +MOVJ EC00165
SMOVL C00166 +MOVJ EC00166
SMOVL C00167 +MOVJ EC00167
SMOVL C00168 +MOVJ EC00168
SMOVL C00169 +MOVJ EC00169
SMOVL C00170 +MOVJ EC00170
SMOVL C00171 +MOVJ EC00171
SMOVL C00172 +MOVJ EC00172
SMOVL C00173 +MOVJ EC00173
SMOVL C00174 +MOVJ EC00174
SMOVL C00175 +MOVJ EC00175
SMOVL C00176 +MOVJ EC00176
SMOVL C00177 +MOVJ EC00177
SMOVL C00178 +MOVJ EC00178
SMOVL C00179 +MOVJ EC00179
SMOVL C00180 +MOVJ EC00180
SMOVL C00181 +MOVJ EC00181
SMOVL C00182 +MOVJ EC00182
SMOVL C00183 +MOVJ EC00183
SMOVL C00184 +MOVJ EC00184
SMOVL C00185 +MOVJ EC00185
SMOVL C00186 +MOVJ EC00186
SMOVL C00187 +MOVJ EC00187
SMOVL C00188 +MOVJ EC00188
SMOVL C00189 +MOVJ EC00189
SMOVL C00190 +MOVJ EC00190
SMOVL C00191 +MOVJ EC00191
SMOVL C00192 +MOVJ EC00192
SMOVL C00193 +MOVJ EC00193
SMOVL C00194 +MOVJ EC00194
SMOVL C00195 +MOVJ EC00195
SMOVL C00196 +MOVJ EC00196
SMOVL C00197 +MOVJ EC00197
SMOVL C00198 +MOVJ EC00198
SMOVL C00199 +MOVJ EC00199
SMOVL C00200 +MOVJ EC00200
SMOVL C00201 +MOVJ EC00201
SMOVL C00202 +MOVJ EC00202
SMOVL C00203 +MOVJ EC00203
SMOVL C00204 +MOVJ EC00204
SMOVL C00205 +MOVJ EC00205
SMOVL C00206 +MOVJ EC00206
SMOVL C00207 +MOVJ EC00207
SMOVL C00208 +MOVJ EC00208
SMOVL C00209 +MOVJ EC00209
SMOVL C00210 +MOVJ EC00210
SMOVL C00211 +MOVJ EC00211
SMOVL C00212 +MOVJ EC00212
SMOVL C00213 +MOVJ EC00213
SMOVL C00214 +MOVJ EC00214
SMOVL C00215 +MOVJ EC00215
SMOVL C00216 +MOVJ EC00216
SMOVL C00217 +MOVJ EC00217
SMOVL C00218 +MOVJ EC00218
SMOVL C00219 +MOVJ EC00219
SMOVL C00220 +MOVJ EC00220
SMOVL C00221 +MOVJ EC00221
SMOVL C00222 +MOVJ EC00222
SMOVL C00223 +MOVJ EC00223
SMOVL C00224 +MOVJ EC00224
SMOVL C00225 +MOVJ EC00225
SMOVL C00226 +MOVJ EC00226
SMOVL C00227 +MOVJ EC00227
SMOVL C00228 +MOVJ EC00228
SMOVL C00229 +MOVJ EC00229
SMOVL C00230 +MOVJ EC00230
SMOVL C00231 +MOVJ EC00231
SMOVL C00232 +MOVJ EC00232
SMOVL C00233 +MOVJ EC00233
SMOVL C00234 +MOVJ EC00234
SMOVL C00235 +MOVJ EC00235
SMOVL C00236 +MOVJ EC00236
SMOVL C00237 +MOVJ EC00237
SMOVL C00238 +MOVJ EC00238
SMOVL C00239 +MOVJ EC00239
SMOVL C00240 +MOVJ EC00240
SMOVL C00241 +MOVJ EC00241
SMOVL C00242 +MOVJ EC00242
SMOVL C00243 +MOVJ EC00243
SMOVL C00244 +MOVJ EC00244
SMOVL C00245 +MOVJ EC00245
SMOVL C00246 +MOVJ EC00246
SMOVL C00247 +MOVJ EC00247
SMOVL C00248 +MOVJ EC00248
SMOVL C00249 +MOVJ EC00249
SMOVL C00250 +MOVJ EC00250
SMOVL C00251 +MOVJ EC00251
SMOVL C00252 +MOVJ EC00252
SMOVL C00253 +MOVJ EC00253
SMOVL C00254 +MOVJ EC00254
SMOVL C00255 +MOVJ EC00255
SMOVL C00256 +MOVJ EC00256
SMOVL C00257 +MOVJ EC00257
SMOVL C00258 +MOVJ EC00258
SMOVL C00259 +MOVJ EC00259
SMOVL C00260 +MOVJ EC00260
SMOVL C00261 +MOVJ EC00261
SMOVL C00262 +MOVJ EC00262
SMOVL C00263 +MOVJ EC00263
SMOVL C00264 +MOVJ EC00264
SMOVL C00265 +MOVJ EC00265
SMOVL C00266 +MOVJ EC00266
SMOVL C00267 +MOVJ EC00267
SMOVL C00268 +MOVJ EC00268
SMOVL C00269 +MOVJ EC00269
SMOVL C00270 +MOVJ EC00270
SMOVL C00271 +MOVJ EC00271
SMOVL C00272 +MOVJ EC00272
SMOVL C00273 +MOVJ EC00273
SMOVL C00274 +MOVJ EC00274
SMOVL C00275 +MOVJ EC00275
SMOVL C00276 +MOVJ EC00276
SMOVL C00277 +MOVJ EC00277
SMOVL C00278 +MOVJ EC00278
SMOVL C00279 +MOVJ EC00279
SMOVL C00280 +MOVJ EC00280
SMOVL C00281 +MOVJ EC00281
SMOVL C00282 +MOVJ EC00282
SMOVL C00283 +MOVJ EC00283
SMOVL C00284 +MOVJ EC00284
SMOVL C00285 +MOVJ EC00285
SMOVL C00286 +MOVJ EC00286
SMOVL C00287 +MOVJ EC00287
SMOVL C00288 +MOVJ EC00288
SMOVL C00289 +MOVJ EC00289
SMOVL C00290 +MOVJ EC00290
SMOVL C00291 +MOVJ EC00291
SMOVL C00292 +MOVJ EC00292
SMOVL C00293 +MOVJ EC00293
SMOVL C00294 +MOVJ EC00294
SMOVL C00295 +MOVJ EC00295
SMOVL C00296 +MOVJ EC00296
SMOVL C00297 +MOVJ EC00297
SMOVL C00298 +MOVJ EC00298
SMOVL C00299 +MOVJ EC00299
SMOVL C00300 +MOVJ EC00300
SMOVL C00301 +MOVJ EC00301
SMOVL C00302 +MOVJ EC00302
SMOVL C00303 +MOVJ EC00303
SMOVL C00304 +MOVJ EC00304
SMOVL C00305 +MOVJ EC00305
SMOVL C00306 +MOVJ EC00306
SMOVL C00307 +MOVJ EC00307
SMOVL C00308 +MOVJ EC00308
SMOVL C00309 +MOVJ EC00309
SMOVL C00310 +MOVJ EC00310
SMOVL C00311 +MOVJ EC00311
SMOVL C00312 +MOVJ EC00312
SMOVL C00313 +MOVJ EC00313
SMOVL C00314 +MOVJ EC00314
SMOVL C00315 +MOVJ EC00315
SMOVL C00316 +MOVJ EC00316
SMOVL C00317 +MOVJ EC00317
SMOVL C00318 +MOVJ EC00318
SMOVL C00319 +MOVJ EC00319
SMOVL C00320 +MOVJ EC00320
SMOVL C00321 +MOVJ EC00321
SMOVL C00322 +MOVJ EC00322
SMOVL C00323 +MOVJ EC00323
SMOVL C00324 +MOVJ EC00324
SMOVL C00325 +MOVJ EC00325
SMOVL C00326 +MOVJ EC00326
SMOVL C00327 +MOVJ EC00327
SMOVL C00328 +MOVJ EC00328
SMOVL C00329 +MOVJ EC00329
SMOVL C00330 +MOVJ EC00330
SMOVL C00331 +MOVJ EC00331
SMOVL C00332 +MOVJ EC00332
SMOVL C00333 +MOVJ EC00333
SMOVL C00334 +MOVJ EC00334
SMOVL C00335 +MOVJ EC00335
SMOVL C00336 +MOVJ EC00336
SMOVL C00337 +MOVJ EC00337
SMOVL C00338 +MOVJ EC00338
SMOVL C00339 +MOVJ EC00339
SMOVL C00340 +MOVJ EC00340
SMOVL C00341 +MOVJ EC00341
SMOVL C00342 +MOVJ EC00342
SMOVL C00343 +MOVJ EC00343
SMOVL C00344 +MOVJ EC00344
SMOVL C00345 +MOVJ EC00345
SMOVL C00346 +MOVJ EC00346
SMOVL C00347 +MOVJ EC00347
SMOVL C00348 +MOVJ EC00348
SMOVL C00349 +MOVJ EC00349
SMOVL C00350 +MOVJ EC00350
SMOVL C00351 +MOVJ EC00351
SMOVL C00352 +MOVJ EC00352
SMOVL C00353 +MOVJ EC00353
SMOVL C00354 +MOVJ EC00354
SMOVL C00355 +MOVJ EC00355
SMOVL C00356 +MOVJ EC00356
SMOVL C00357 +MOVJ EC00357
SMOVL C00358 +MOVJ EC00358
SMOVL C00359 +MOVJ EC00359
SMOVL C00360 +MOVJ EC00360
SMOVL C00361 +MOVJ EC00361
SMOVL C00362 +MOVJ EC00362
SMOVL C00363 +MOVJ EC00363
SMOVL C00364 +MOVJ EC00364
SMOVL C00365 +MOVJ EC00365
SMOVL C00366 +MOVJ EC00366
SMOVL C00367 +MOVJ EC00367
SMOVL C00368 +MOVJ EC00368
SMOVL C00369 +MOVJ EC00369
SMOVL C00370 +MOVJ EC00370
SMOVL C00371 +MOVJ EC00371
SMOVL C00372 +MOVJ EC00372
SMOVL C00373 +MOVJ EC00373
SMOVL C00374 +MOVJ EC00374
SMOVL C00375 +MOVJ EC00375
SMOVL C00376 +MOVJ EC00376
SMOVL C00377 +MOVJ EC00377
SMOVL C00378 +MOVJ EC00378
SMOVL C00379 +MOVJ EC00379
SMOVL C00380 +MOVJ EC00380
SMOVL C00381 +MOVJ EC00381
SMOVL C00382 +MOVJ EC00382
SMOVL C00383 +MOVJ EC00383
SMOVL C00384 +MOVJ EC00384
SMOVL C00385 +MOVJ EC00385
SMOVL C00386 +MOVJ EC00386
SMOVL C00387 +MOVJ EC00387
SMOVL C00388 +MOVJ EC00388
SMOVL C00389 +MOVJ EC00389
SMOVL C00390 +MOVJ EC00390
SMOVL C00391 +MOVJ EC00391
SMOVL C00392 +MOVJ EC00392
SMOVL C00393 +MOVJ EC00393
SMOVL C00394 +MOVJ EC00394
SMOVL C00395 +MOVJ EC00395
SMOVL C00396 +MOVJ EC00396
SMOVL C00397 +MOVJ EC00397
SMOVL C00398 +MOVJ EC00398
SMOVL C00399 +MOVJ EC00399
SMOVL C00400 +MOVJ EC00400
SMOVL C00401 +MOVJ EC00401
SMOVL C00402 +MOVJ EC00402
SMOVL C00403 +MOVJ EC00403
SMOVL C00404 +MOVJ EC00404
SMOVL C00405 +MOVJ EC00405
SMOVL C00406 +MOVJ EC00406
SMOVL C00407 +MOVJ EC00407
SMOVL C00408 +MOVJ EC00408
SMOVL C00409 +MOVJ EC00409
SMOVL C00410 +MOVJ EC00410
SMOVL C00411 +MOVJ EC00411
SMOVL C00412 +MOVJ EC00412
SMOVL C00413 +MOVJ EC00413
SMOVL C00414 +MOVJ EC00414
SMOVL C00415 +MOVJ EC00415
SMOVL C00416 +MOVJ EC00416
SMOVL C00417 +MOVJ EC00417
SMOVL C00418 +MOVJ EC00418
SMOVL C00419 +MOVJ EC00419
SMOVL C00420 +MOVJ EC00420
SMOVL C00421 +MOVJ EC00421
SMOVL C00422 +MOVJ EC00422
SMOVL C00423 +MOVJ EC00423
SMOVL C00424 +MOVJ EC00424
SMOVL C00425 +MOVJ EC00425
SMOVL C00426 +MOVJ EC00426
SMOVL C00427 +MOVJ EC00427
SMOVL C00428 +MOVJ EC00428
SMOVL C00429 +MOVJ EC00429
SMOVL C00430 +MOVJ EC00430
SMOVL C00431 +MOVJ EC00431
SMOVL C00432 +MOVJ EC00432
SMOVL C00433 +MOVJ EC00433
SMOVL C00434 +MOVJ EC00434
SMOVL C00435 +MOVJ EC00435
SMOVL C00436 +MOVJ EC00436
SMOVL C00437 +MOVJ EC00437
SMOVL C00438 +MOVJ EC00438
SMOVL C00439 +MOVJ EC00439
SMOVL C00440 +MOVJ EC00440
SMOVL C00441 +MOVJ EC00441
SMOVL C00442 +MOVJ EC00442
SMOVL C00443 +MOVJ EC00443
SMOVL C00444 +MOVJ EC00444
SMOVL C00445 +MOVJ EC00445
SMOVL C00446 +MOVJ EC00446
SMOVL C00447 +MOVJ EC00447
SMOVL C00448 +MOVJ EC00448
SMOVL C00449 +MOVJ EC00449
SMOVL C00450 +MOVJ EC00450
SMOVL C00451 +MOVJ EC00451
SMOVL C00452 +MOVJ EC00452
SMOVL C00453 +MOVJ EC00453
SMOVL C00454 +MOVJ EC00454
SMOVL C00455 +MOVJ EC00455
SMOVL C00456 +MOVJ EC00456
SMOVL C00457 +MOVJ EC00457
SMOVL C00458 +MOVJ EC00458
SMOVL C00459 +MOVJ EC00459
SMOVL C00460 +MOVJ EC00460
SMOVL C00461 +MOVJ EC00461
SMOVL C00462 +MOVJ EC00462
SMOVL C00463 +MOVJ EC00463
SMOVL C00464 +MOVJ EC00464
SMOVL C00465 +MOVJ EC00465
SMOVL C00466 +MOVJ EC00466
SMOVL C00467 +MOVJ EC00467
SMOVL C00468 +MOVJ EC00468
SMOVL C00469 +MOVJ EC00469
SMOVL C00470 +MOVJ EC00470
SMOVL C00471 +MOVJ EC00471
SMOVL C00472 +MOVJ EC00472
SMOVL C00473 +MOVJ EC00473
SMOVL C00474 +MOVJ EC00474
SMOVL C00475 +MOVJ EC00475
SMOVL C00476 +MOVJ EC00476
SMOVL C00477 +MOVJ EC00477
SMOVL C00478 +MOVJ EC00478
SMOVL C00479 +MOVJ EC00479
SMOVL C00480 +MOVJ EC00480
SMOVL C00481 +MOVJ EC00481
SMOVL C00482 +MOVJ EC00482
SMOVL C00483 +MOVJ EC00483
SMOVL C00484 +MOVJ EC00484
SMOVL C00485 +MOVJ EC00485
SMOVL C00486 +MOVJ EC00486
SMOVL C00487 +MOVJ EC00487
SMOVL C00488 +MOVJ EC00488
SMOVL C00489 +MOVJ EC00489
SMOVL C00490 +MOVJ EC00490
SMOVL C00491 +MOVJ EC00491
SMOVL C00492 +MOVJ EC00492
SMOVL C00493 +MOVJ EC00493
SMOVL C00494 +MOVJ EC00494
SMOVL C00495 +MOVJ EC00495
SMOVL C00496 +MOVJ EC00496
SMOVL C00497 +MOVJ EC00497
SMOVL C00498 +MOVJ EC00498
SMOVL C00499 +MOVJ EC00499
SMOVL C00500 +MOVJ EC00500
SMOVL C00501 +MOVJ EC00501
SMOVL C00502 +MOVJ EC00502
SMOVL C00503 +MOVJ EC00503
SMOVL C00504 +MOVJ EC00504
SMOVL C00505 +MOVJ EC00505
SMOVL C00506 +MOVJ EC00506
SMOVL C00507 +MOVJ EC00507
SMOVL C00508 +MOVJ EC00508
SMOVL C00509 +MOVJ EC00509
SMOVL C00510 +MOVJ EC00510
SMOVL C00511 +MOVJ EC00511
SMOVL C00512 +MOVJ EC00512
SMOVL C00513 +MOVJ EC00513
SMOVL C00514 +MOVJ EC00514
SMOVL C00515 +MOVJ EC00515
SMOVL C00516 +MOVJ EC00516
SMOVL C00517 +MOVJ EC00517
SMOVL C00518 +MOVJ EC00518
SMOVL C00519 +MOVJ EC00519
SMOVL C00520 +MOVJ EC00520
SMOVL C00521 +MOVJ EC00521
SMOVL C00522 +MOVJ EC00522
SMOVL C00523 +MOVJ EC00523
SMOVL C00524 +MOVJ EC00524
SMOVL C00525 +MOVJ EC00525
SMOVL C00526 +MOVJ EC00526
SMOVL C00527 +MOVJ EC00527
SMOVL C00528 +MOVJ EC00528
SMOVL C00529 +MOVJ EC00529
SMOVL C00530 +MOVJ EC00530
SMOVL C00531 +MOVJ EC00531
SMOVL C00532 +MOVJ EC00532
SMOVL C00533 +MOVJ EC00533
SMOVL C00534 +MOVJ EC00534
SMOVL C00535 +MOVJ EC00535
SMOVL C00536 +MOVJ EC00536
SMOVL C00537 +MOVJ EC00537
SMOVL C00538 +MOVJ EC00538
SMOVL C00539 +MOVJ EC00539
SMOVL C00540 +MOVJ EC00540
SMOVL C00541 +MOVJ EC00541
SMOVL C00542 +MOVJ EC00542
SMOVL C00543 +MOVJ EC00543
SMOVL C00544 +MOVJ EC00544
SMOVL C00545 +MOVJ EC00545
SMOVL C00546 +MOVJ EC00546
SMOVL C00547 +MOVJ EC00547
SMOVL C00548 +MOVJ EC00548
SMOVL C00549 +MOVJ EC00549
SMOVL C00550 +MOVJ EC00550
SMOVL C00551 +MOVJ EC00551
SMOVL C00552 +MOVJ EC00552
SMOVL C00553 +MOVJ EC00553
SMOVL C00554 +MOVJ EC00554
SMOVL C00555 +MOVJ EC00555
SMOVL C00556 +MOVJ EC00556
SMOVL C00557 +MOVJ EC00557
SMOVL C00558 +MOVJ EC00558
SMOVL C00559 +MOVJ EC00559
SMOVL C00560 +MOVJ EC00560
SMOVL C00561 +MOVJ EC00561
SMOVL C00562 +MOVJ EC00562
SMOVL C00563 +MOVJ EC00563
SMOVL C00564 +MOVJ EC00564
SMOVL C00565 +MOVJ EC00565
SMOVL C00566 +MOVJ EC00566
SMOVL C00567 +MOVJ EC00567
SMOVL C00568 +MOVJ EC00568
SMOVL C00569 +MOVJ EC00569
SMOVL C00570 +MOVJ EC00570
SMOVL C00571 +MOVJ EC00571
SMOVL C00572 +MOVJ EC00572
SMOVL C00573 +MOVJ EC00573
SMOVL C00574 +MOVJ EC00574
SMOVL C00575 +MOVJ EC00575
SMOVL C00576 +MOVJ EC00576
SMOVL C00577 +MOVJ EC00577
SMOVL C00578 +MOVJ EC00578
SMOVL C00579 +MOVJ EC00579
SMOVL C00580 +MOVJ EC00580
SMOVL C00581 +MOVJ EC00581
SMOVL C00582 +MOVJ EC00582
SMOVL C00583 +MOVJ EC00583
SMOVL C00584 +MOVJ EC00584
SMOVL C00585 +MOVJ EC00585
SMOVL C00586 +MOVJ EC00586
SMOVL C00587 +MOVJ EC00587
SMOVL C00588 +MOVJ EC00588
SMOVL C00589 +MOVJ EC00589
SMOVL C00590 +MOVJ EC00590
SMOVL C00591 +MOVJ EC00591
SMOVL C00592 +MOVJ EC00592
SMOVL C00593 +MOVJ EC00593
SMOVL C00594 +MOVJ EC00594
SMOVL C00595 +MOVJ EC00595
SMOVL C00596 +MOVJ EC00596
SMOVL C00597 +MOVJ EC00597
SMOVL C00598 +MOVJ EC00598
SMOVL C00599 +MOVJ EC00599
SMOVL C00600 +MOVJ EC00600
SMOVL C00601 +MOVJ EC00601
SMOVL C00602 +MOVJ EC00602
SMOVL C00603 +MOVJ EC00603
SMOVL C00604 +MOVJ EC00604
SMOVL C00605 +MOVJ EC00605
SMOVL C00606 +MOVJ EC00606
SMOVL C00607 +MOVJ EC00607
SMOVL C00608 +MOVJ EC00608
SMOVL C00609 +MOVJ EC00609
SMOVL C00610 +MOVJ EC00610
SMOVL C00611 +MOVJ EC00611
SMOVL C00612 +MOVJ EC00612
SMOVL C00613 +MOVJ EC00613
SMOVL C00614 +MOVJ EC00614
SMOVL C00615 +MOVJ EC00615
SMOVL C00616 +MOVJ EC00616
SMOVL C00617 +MOVJ EC00617
SMOVL C00618 +MOVJ EC00618
SMOVL C00619 +MOVJ EC00619
SMOVL C00620 +MOVJ EC00620
SMOVL C00621 +MOVJ EC00621
SMOVL C00622 +MOVJ EC00622
SMOVL C00623 +MOVJ EC00623
SMOVL C00624 +MOVJ EC00624
SMOVL C00625 +MOVJ EC00625
SMOVL C00626 +MOVJ EC00626
SMOVL C00627 +MOVJ EC00627
SMOVL C00628 +MOVJ EC00628
SMOVL C00629 +MOVJ EC00629
SMOVL C00630 +MOVJ EC00630
SMOVL C00631 +MOVJ EC00631
SMOVL C00632 +MOVJ EC00632
SMOVL C00633 +MOVJ EC00633
SMOVL C00634 +MOVJ EC00634
SMOVL C00635 +MOVJ EC00635
SMOVL C00636 +MOVJ EC00636
SMOVL C00637 +MOVJ EC00637
SMOVL C00638 +MOVJ EC00638
SMOVL C00639 +MOVJ EC00639
SMOVL C00640 +MOVJ EC00640
SMOVL C00641 +MOVJ EC00641
SMOVL C00642 +MOVJ EC00642
SMOVL C00643 +MOVJ EC00643
SMOVL C00644 +MOVJ EC00644
SMOVL C00645 +MOVJ EC00645
SMOVL C00646 +MOVJ EC00646
SMOVL C00647 +MOVJ EC00647
SMOVL C00648 +MOVJ EC00648
SMOVL C00649 +MOVJ EC00649
SMOVL C00650 +MOVJ EC00650
SMOVL C00651 +MOVJ EC00651
SMOVL C00652 +MOVJ EC00652
SMOVL C00653 +MOVJ EC00653
SMOVL C00654 +MOVJ EC00654
SMOVL C00655 +MOVJ EC00655
SMOVL C00656 +MOVJ EC00656
SMOVL C00657 +MOVJ EC00657
SMOVL C00658 +MOVJ EC00658
SMOVL C00659 +MOVJ EC00659
SMOVL C00660 +MOVJ EC00660
SMOVL C00661 +MOVJ EC00661
SMOVL C00662 +MOVJ EC00662
SMOVL C00663 +MOVJ EC00663
SMOVL C00664 +MOVJ EC00664
SMOVL C00665 +MOVJ EC00665
SMOVL C00666 +MOVJ EC00666
SMOVL C00667 +MOVJ EC00667
SMOVL C00668 +MOVJ EC00668
SMOVL C00669 +MOVJ EC00669
SMOVL C00670 +MOVJ EC00670
SMOVL C00671 +MOVJ EC00671
SMOVL C00672 +MOVJ EC00672
SMOVL C00673 +MOVJ EC00673
SMOVL C00674 +MOVJ EC00674
SMOVL C00675 +MOVJ EC00675
SMOVL C00676 +MOVJ EC00676
SMOVL C00677 +MOVJ EC00677
SMOVL C00678 +MOVJ EC00678
SMOVL C00679 +MOVJ EC00679
SMOVL C00680 +MOVJ EC00680
SMOVL C00681 +MOVJ EC00681
SMOVL C00682 +MOVJ EC00682
SMOVL C00683 +MOVJ EC00683
SMOVL C00684 +MOVJ EC00684
SMOVL C00685 +MOVJ EC00685
SMOVL C00686 +MOVJ EC00686
SMOVL C00687 +MOVJ EC00687
SMOVL C00688 +MOVJ EC00688
SMOVL C00689 +MOVJ EC00689
SMOVL C00690 +MOVJ EC00690
SMOVL C00691 +MOVJ EC00691
SMOVL C00692 +MOVJ EC00692
SMOVL C00693 +MOVJ EC00693
SMOVL C00694 +MOVJ EC00694
SMOVL C00695 +MOVJ EC00695
SMOVL C00696 +MOVJ EC00696
SMOVL C00697 +MOVJ EC00697
SMOVL C00698 +MOVJ EC00698
SMOVL C00699 +MOVJ EC00699
SMOVL C00700 +MOVJ EC00700
SMOVL C00701 +MOVJ EC00701
SMOVL C00702 +MOVJ EC00702
SMOVL C00703 +MOVJ EC00703
SMOVL C00704 +MOVJ EC00704
SMOVL C00705 +MOVJ EC00705
SMOVL C00706 +MOVJ EC00706
SMOVL C00707 +MOVJ EC00707
SMOVL C00708 +MOVJ EC00708
SMOVL C00709 +MOVJ EC00709
SMOVL C00710 +MOVJ EC00710
SMOVL C00711 +MOVJ EC00711
SMOVL C00712 +MOVJ EC00712
SMOVL C00713 +MOVJ EC00713
SMOVL C00714 +MOVJ EC00714
SMOVL C00715 +MOVJ EC00715
SMOVL C00716 +MOVJ EC00716
SMOVL C00717 +MOVJ EC00717
SMOVL C00718 +MOVJ EC00718
SMOVL C00719 +MOVJ EC00719
SMOVL C00720 +MOVJ EC00720
SMOVL C00721 +MOVJ EC00721
SMOVL C00722 +MOVJ EC00722
SMOVL C00723 +MOVJ EC00723
SMOVL C00724 +MOVJ EC00724
SMOVL C00725 +MOVJ EC00725
SMOVL C00726 +MOVJ EC00726
SMOVL C00727 +MOVJ EC00727
SMOVL C00728 +MOVJ EC00728
SMOVL C00729 +MOVJ EC00729
SMOVL C00730 +MOVJ EC00730
SMOVL C00731 +MOVJ EC00731
SMOVL C00732 +MOVJ EC00732
SMOVL C00733 +MOVJ EC00733
SMOVL C00734 +MOVJ EC00734
SMOVL C00735 +MOVJ EC00735
SMOVL C00736 +MOVJ EC00736
SMOVL C00737 +MOVJ EC00737
SMOVL C00738 +MOVJ EC00738
SMOVL C00739 +MOVJ EC00739
SMOVL C00740 +MOVJ EC00740
SMOVL C00741 +MOVJ EC00741
SMOVL C00742 +MOVJ EC00742
SMOVL C00743 +MOVJ EC00743
SMOVL C00744 +MOVJ EC00744
SMOVL C00745 +MOVJ EC00745
SMOVL C00746 +MOVJ EC00746
SMOVL C00747 +MOVJ EC00747
SMOVL C00748 +MOVJ EC00748
SMOVL C00749 +MOVJ EC00749
SMOVL C00750 +MOVJ EC00750
SMOVL C00751 +MOVJ EC00751
SMOVL C00752 +MOVJ EC00752
SMOVL C00753 +MOVJ EC00753
SMOVL C00754 +MOVJ EC00754
SMOVL C00755 +MOVJ EC00755
SMOVL C00756 +MOVJ EC00756
SMOVL C00757 +MOVJ EC00757
SMOVL C00758 +MOVJ EC00758
SMOVL C00759 +MOVJ EC00759
SMOVL C00760 +MOVJ EC00760
SMOVL C00761 +MOVJ EC00761
SMOVL C00762 +MOVJ EC00762
SMOVL C00763 +MOVJ EC00763
SMOVL C00764 +MOVJ EC00764
SMOVL C00765 +MOVJ EC00765
SMOVL C00766 +MOVJ EC00766
SMOVL C00767 +MOVJ EC00767
SMOVL C00768 +MOVJ EC00768
SMOVL C00769 +MOVJ EC00769
SMOVL C00770 +MOVJ EC00770
SMOVL C00771 +MOVJ EC00771
SMOVL C00772 +MOVJ EC00772
SMOVL C00773 +MOVJ EC00773
SMOVL C00774 +MOVJ EC00774
SMOVL C00775 +MOVJ EC00775
SMOVL C00776 +MOVJ EC00776
SMOVL C00777 +MOVJ EC00777
SMOVL C00778 +MOVJ EC00778
SMOVL C00779 +MOVJ EC00779
SMOVL C00780 +MOVJ EC00780
SMOVL C00781 +MOVJ EC00781
SMOVL C00782 +MOVJ EC00782
SMOVL C00783 +MOVJ EC00783
SMOVL C00784 +MOVJ EC00784
SMOVL C00785 +MOVJ EC00785
SMOVL C00786 +MOVJ EC00786
SMOVL C00787 +MOVJ EC00787
SMOVL C00788 +MOVJ EC00788
SMOVL C00789 +MOVJ EC00789
SMOVL C00790 +MOVJ EC00790
SMOVL C00791 +MOVJ EC00791
SMOVL C00792 +MOVJ EC00792
SMOVL C00793 +MOVJ EC00793
SMOVL C00794 +MOVJ EC00794
SMOVL C00795 +MOVJ EC00795
SMOVL C00796 +MOVJ EC00796
SMOVL C00797 +MOVJ EC00797
SMOVL C00798 +MOVJ EC00798
SMOVL C00799 +MOVJ EC00799
SMOVL C00800 +MOVJ EC00800
SMOVL C00801 +MOVJ EC00801
SMOVL C00802 +MOVJ EC00802
SMOVL C00803 +MOVJ EC00803
SMOVL C00804 +MOVJ EC00804
SMOVL C00805 +MOVJ EC00805
SMOVL C00806 +MOVJ EC00806
SMOVL C00807 +MOVJ EC00807
SMOVL C00808 +MOVJ EC00808
SMOVL C00809 +MOVJ EC00809
SMOVL C00810 +MOVJ EC00810
SMOVL C00811 +MOVJ EC00811
SMOVL C00812 +MOVJ EC00812
SMOVL C00813 +MOVJ EC00813
SMOVL C00814 +MOVJ EC00814
SMOVL C00815 +MOVJ EC00815
SMOVL C00816 +MOVJ EC00816
SMOVL C00817 +MOVJ EC00817
SMOVL C00818 +MOVJ EC00818
SMOVL C00819 +MOVJ EC00819
SMOVL C00820 +MOVJ EC00820
SMOVL C00821 +MOVJ EC00821
SMOVL C00822 +MOVJ EC00822
SMOVL C00823 +MOVJ EC00823
SMOVL C00824 +MOVJ EC00824
SMOVL C00825 +MOVJ EC00825
SMOVL C00826 +MOVJ EC00826
SMOVL C00827 +MOVJ EC00827
SMOVL C00828 +MOVJ EC00828
SMOVL C00829 +MOVJ EC00829
SMOVL C00830 +MOVJ EC00830
SMOVL C00831 +MOVJ EC00831
SMOVL C00832 +MOVJ EC00832
SMOVL C00833 +MOVJ EC00833
SMOVL C00834 +MOVJ EC00834
SMOVL C00835 +MOVJ EC00835
SMOVL C00836 +MOVJ EC00836
SMOVL C00837 +MOVJ EC00837
SMOVL C00838 +MOVJ EC00838
SMOVL C00839 +MOVJ EC00839
SMOVL C00840 +MOVJ EC00840
SMOVL C00841 +MOVJ EC00841
SMOVL C00842 +MOVJ EC00842
SMOVL C00843 +MOVJ EC00843
SMOVL C00844 +MOVJ EC00844
SMOVL C00845 +MOVJ EC00845
SMOVL C00846 +MOVJ EC00846
SMOVL C00847 +MOVJ EC00847
SMOVL C00848 +MOVJ EC00848
SMOVL C00849 +MOVJ EC00849
SMOVL C00850 +MOVJ EC00850
SMOVL C00851 +MOVJ EC00851
SMOVL C00852 +MOVJ EC00852
SMOVL C00853 +MOVJ EC00853
SMOVL C00854 +MOVJ EC00854
SMOVL C00855 +MOVJ EC00855
SMOVL C00856 +MOVJ EC00856
SMOVL C00857 +MOVJ EC00857
SMOVL C00858 +MOVJ EC00858
SMOVL C00859 +MOVJ EC00859
SMOVL C00860 +MOVJ EC00860
SMOVL C00861 +MOVJ EC00861
SMOVL C00862 +MOVJ EC00862
SMOVL C00863 +MOVJ EC00863
SMOVL C00864 +MOVJ EC00864
SMOVL C00865 +MOVJ EC00865
SMOVL C00866 +MOVJ EC00866
SMOVL C00867 +MOVJ EC00867
SMOVL C00868 +MOVJ EC00868
SMOVL C00869 +MOVJ EC00869
SMOVL C00870 +MOVJ EC00870
SMOVL C00871 +MOVJ EC00871
SMOVL C00872 +MOVJ EC00872
SMOVL C00873 +MOVJ EC00873
SMOVL C00874 +MOVJ EC00874
SMOVL C00875 +MOVJ EC00875
SMOVL C00876 +MOVJ EC00876
SMOVL C00877 +MOVJ EC00877
SMOVL C00878 +MOVJ EC00878
SMOVL C00879 +MOVJ EC00879
SMOVL C00880 +MOVJ EC00880
SMOVL C00881 +MOVJ EC00881
SMOVL C00882 +MOVJ EC00882
SMOVL C00883 +MOVJ EC00883
SMOVL C00884 +MOVJ EC00884
SMOVL C00885 +MOVJ EC00885
SMOVL C00886 +MOVJ EC00886
SMOVL C00887 +MOVJ EC00887
SMOVL C00888 +MOVJ EC00888
SMOVL C00889 +MOVJ EC00889
SMOVL C00890 +MOVJ EC00890
SMOVL C00891 +MOVJ EC00891
SMOVL C00892 +MOVJ EC00892
SMOVL C00893 +MOVJ EC00893
SMOVL C00894 +MOVJ EC00894
SMOVL C00895 +MOVJ EC00895
SMOVL C00896 +MOVJ EC00896
SMOVL C00897 +MOVJ EC00897
SMOVL C00898 +MOVJ EC00898
SMOVL C00899 +MOVJ EC00899
SMOVL C00900 +MOVJ EC00900
SMOVL C00901 +MOVJ EC00901
SMOVL C00902 +MOVJ EC00902
SMOVL C00903 +MOVJ EC00903
SMOVL C00904 +MOVJ EC00904
SMOVL C00905 +MOVJ EC00905
SMOVL C00906 +MOVJ EC00906
SMOVL C00907 +MOVJ EC00907
SMOVL C00908 +MOVJ EC00908
SMOVL C00909 +MOVJ EC00909
SMOVL C00910 +MOVJ EC00910
SMOVL C00911 +MOVJ EC00911
SMOVL C00912 +MOVJ EC00912
SMOVL C00913 +MOVJ EC00913
SMOVL C00914 +MOVJ EC00914
SMOVL C00915 +MOVJ EC00915
SMOVL C00916 +MOVJ EC00916
SMOVL C00917 +MOVJ EC00917
SMOVL C00918 +MOVJ EC00918
SMOVL C00919 +MOVJ EC00919
SMOVL C00920 +MOVJ EC00920
SMOVL C00921 +MOVJ EC00921
SMOVL C00922 +MOVJ EC00922
SMOVL C00923 +MOVJ EC00923
SMOVL C00924 +MOVJ EC00924
SMOVL C00925 +MOVJ EC00925
SMOVL C00926 +MOVJ EC00926
SMOVL C00927 +MOVJ EC00927
SMOVL C00928 +MOVJ EC00928
SMOVL C00929 +MOVJ EC00929
SMOVL C00930 +MOVJ EC00930
SMOVL C00931 +MOVJ EC00931
SMOVL C00932 +MOVJ EC00932
SMOVL C00933 +MOVJ EC00933
SMOVL C00934 +MOVJ EC00934
SMOVL C00935 +MOVJ EC00935
SMOVL C00936 +MOVJ EC00936
SMOVL C00937 +MOVJ EC00937
SMOVL C00938 +MOVJ EC00938
SMOVL C00939 +MOVJ EC00939
SMOVL C00940 +MOVJ EC00940
SMOVL C00941 +MOVJ EC00941
SMOVL C00942 +MOVJ EC00942
SMOVL C00943 +MOVJ EC00943
SMOVL C00944 +MOVJ EC00944
SMOVL C00945 +MOVJ EC00945
SMOVL C00946 +MOVJ EC00946
SMOVL C00947 +MOVJ EC00947
SMOVL C00948 +MOVJ EC00948
SMOVL C00949 +MOVJ EC00949
SMOVL C00950 +MOVJ EC00950
SMOVL C00951 +MOVJ EC00951
SMOVL C00952 +MOVJ EC00952
SMOVL C00953 +MOVJ EC00953
SMOVL C00954 +MOVJ EC00954
SMOVL C00955 +MOVJ EC00955
SMOVL C00956 +MOVJ EC00956
SMOVL C00957 +MOVJ EC00957
SMOVL C00958 +MOVJ EC00958
SMOVL C00959 +MOVJ EC00959
SMOVL C00960 +MOVJ EC00960
SMOVL C00961 +MOVJ EC00961
SMOVL C00962 +MOVJ EC00962
SMOVL C00963 +MOVJ EC00963
SMOVL C00964 +MOVJ EC00964
SMOVL C00965 +MOVJ EC00965
SMOVL C00966 +MOVJ EC00966
SMOVL C00967 +MOVJ EC00967
SMOVL C00968 +MOVJ EC00968
SMOVL C00969 +MOVJ EC00969
SMOVL C00970 +MOVJ EC00970
SMOVL C00971 +MOVJ EC00971
SMOVL C00972 +MOVJ EC00972
SMOVL C00973 +MOVJ EC00973
SMOVL C00974 +MOVJ EC00974
SMOVL C00975 +MOVJ EC00975
SMOVL C00976 +MOVJ EC00976
SMOVL C00977 +MOVJ EC00977
SMOVL C00978 +MOVJ EC00978
SMOVL C00979 +MOVJ EC00979
SMOVL C00980 +MOVJ EC00980
SMOVL C00981 +MOVJ EC00981
SMOVL C00982 +MOVJ EC00982
SMOVL C00983 +MOVJ EC00983
SMOVL C00984 +MOVJ EC00984
SMOVL C00985 +MOVJ EC00985
SMOVL C00986 +MOVJ EC00986
SMOVL C00987 +MOVJ EC00987
SMOVL C00988 +MOVJ EC00988
SMOVL C00989 +MOVJ EC00989
SMOVL C00990 +MOVJ EC00990
SMOVL C00991 +MOVJ EC00991
SMOVL C00992 +MOVJ EC00992
SMOVL C00993 +MOVJ EC00993
SMOVL C00994 +MOVJ EC00994
SMOVL C00995 +MOVJ EC00995
SMOVL C00996 +MOVJ EC00996
SMOVL C00997 +MOVJ EC00997
SMOVL C00998 +MOVJ EC00998
SMOVL C00999 +MOVJ EC00999
SMOVL C01000 +MOVJ EC01000
SMOVL C01001 +MOVJ EC01001
SMOVL C01002 +MOVJ EC01002
SMOVL C01003 +MOVJ EC01003
SMOVL C01004 +MOVJ EC01004
SMOVL C01005 +MOVJ EC01005
SMOVL C01006 +MOVJ EC01006
SMOVL C01007 +MOVJ EC01007
SMOVL C01008 +MOVJ EC01008
SMOVL C01009 +MOVJ EC01009
SMOVL C01010 +MOVJ EC01010
SMOVL C01011 +MOVJ EC01011
SMOVL C01012 +MOVJ EC01012
SMOVL C01013 +MOVJ EC01013
SMOVL C01014 +MOVJ EC01014
SMOVL C01015 +MOVJ EC01015
SMOVL C01016 +MOVJ EC01016
SMOVL C01017 +MOVJ EC01017
SMOVL C01018 +MOVJ EC01018
SMOVL C01019 +MOVJ EC01019
SMOVL C01020 +MOVJ EC01020
SMOVL C01021 +MOVJ EC01021
SMOVL C01022 +MOVJ EC01022
SMOVL C01023 +MOVJ EC01023
SMOVL C01024 +MOVJ EC01024
SMOVL C01025 +MOVJ EC01025
SMOVL C01026 +MOVJ EC01026
SMOVL C01027 +MOVJ EC01027
SMOVL C01028 +MOVJ EC01028
SMOVL C01029 +MOVJ EC01029
SMOVL C01030 +MOVJ EC01030
SMOVL C01031 +MOVJ EC01031
SMOVL C01032 +MOVJ EC01032
SMOVL C01033 +MOVJ EC01033
SMOVL C01034 +MOVJ EC01034
SMOVL C01035 +MOVJ EC01035
SMOVL C01036 +MOVJ EC01036
SMOVL C01037 +MOVJ EC01037
SMOVL C01038 +MOVJ EC01038
SMOVL C01039 +MOVJ EC01039
SMOVL C01040 +MOVJ EC01040
SMOVL C01041 +MOVJ EC01041
SMOVL C01042 +MOVJ EC01042
SMOVL C01043 +MOVJ EC01043
SMOVL C01044 +MOVJ EC01044
SMOVL C01045 +MOVJ EC01045
SMOVL C01046 +MOVJ EC01046
SMOVL C01047 +MOVJ EC01047
SMOVL C01048 +MOVJ EC01048
SMOVL C01049 +MOVJ EC01049
SMOVL C01050 +MOVJ EC01050
SMOVL C01051 +MOVJ EC01051
SMOVL C01052 +MOVJ EC01052
SMOVL C01053 +MOVJ EC01053
SMOVL C01054 +MOVJ EC01054
SMOVL C01055 +MOVJ EC01055
SMOVL C01056 +MOVJ EC01056
SMOVL C01057 +MOVJ EC01057
SMOVL C01058 +MOVJ EC01058
SMOVL C01059 +MOVJ EC01059
SMOVL C01060 +MOVJ EC01060
SMOVL C01061 +MOVJ EC01061
SMOVL C01062 +MOVJ EC01062
SMOVL C01063 +MOVJ EC01063
SMOVL C01064 +MOVJ EC01064
SMOVL C01065 +MOVJ EC01065
SMOVL C01066 +MOVJ EC01066
SMOVL C01067 +MOVJ EC01067
SMOVL C01068 +MOVJ EC01068
SMOVL C01069 +MOVJ EC01069
SMOVL C01070 +MOVJ EC01070
SMOVL C01071 +MOVJ EC01071
SMOVL C01072 +MOVJ EC01072
SMOVL C01073 +MOVJ EC01073
SMOVL C01074 +MOVJ EC01074
SMOVL C01075 +MOVJ EC01075
SMOVL C01076 +MOVJ EC01076
SMOVL C01077 +MOVJ EC01077
SMOVL C01078 +MOVJ EC01078
SMOVL C01079 +MOVJ EC01079
SMOVL C01080 +MOVJ EC01080
SMOVL C01081 +MOVJ EC01081
SMOVL C01082 +MOVJ EC01082
SMOVL C01083 +MOVJ EC01083
SMOVL C01084 +MOVJ EC01084
SMOVL C01085 +MOVJ EC01085
SMOVL C01086 +MOVJ EC01086
SMOVL C01087 +MOVJ EC01087
SMOVL C01088 +MOVJ EC01088
SMOVL C01089 +MOVJ EC01089
SMOVL C01090 +MOVJ EC01090
SMOVL C01091 +MOVJ EC01091
SMOVL C01092 +MOVJ EC01092
SMOVL C01093 +MOVJ EC01093
SMOVL C01094 +MOVJ EC01094
SMOVL C01095 +MOVJ EC01095
SMOVL C01096 +MOVJ EC01096
SMOVL C01097 +MOVJ EC01097
SMOVL C01098 +MOVJ EC01098
SMOVL C01099 +MOVJ EC01099
SMOVL C01100 +MOVJ EC01100
SMOVL C01101 +MOVJ EC01101
SMOVL C01102 +MOVJ EC01102
SMOVL C01103 +MOVJ EC01103
SMOVL C01104 +MOVJ EC01104
SMOVL C01105 +MOVJ EC01105
SMOVL C01106 +MOVJ EC01106
SMOVL C01107 +MOVJ EC01107
SMOVL C01108 +MOVJ EC01108
SMOVL C01109 +MOVJ EC01109
SMOVL C01110 +MOVJ EC01110
SMOVL C01111 +MOVJ EC01111
SMOVL C01112 +MOVJ EC01112
SMOVL C01113 +MOVJ EC01113
SMOVL C01114 +MOVJ EC01114
SMOVL C01115 +MOVJ EC01115
SMOVL C01116 +MOVJ EC01116
SMOVL C01117 +MOVJ EC01117
SMOVL C01118 +MOVJ EC01118
SMOVL C01119 +MOVJ EC01119
SMOVL C01120 +MOVJ EC01120
SMOVL C01121 +MOVJ EC01121
SMOVL C01122 +MOVJ EC01122
SMOVL C01123 +MOVJ EC01123
SMOVL C01124 +MOVJ EC01124
SMOVL C01125 +MOVJ EC01125
SMOVL C01126 +MOVJ EC01126
SMOVL C01127 +MOVJ EC01127
SMOVL C01128 +MOVJ EC01128
SMOVL C01129 +MOVJ EC01129
SMOVL C01130 +MOVJ EC01130
SMOVL C01131 +MOVJ EC01131
SMOVL C01132 +MOVJ EC01132
SMOVL C01133 +MOVJ EC01133
SMOVL C01134 +MOVJ EC01134
SMOVL C01135 +MOVJ EC01135
SMOVL C01136 +MOVJ EC01136
SMOVL C01137 +MOVJ EC01137
SMOVL C01138 +MOVJ EC01138
SMOVL C01139 +MOVJ EC01139
SMOVL C01140 +MOVJ EC01140
SMOVL C01141 +MOVJ EC01141
SMOVL C01142 +MOVJ EC01142
SMOVL C01143 +MOVJ EC01143
SMOVL C01144 +MOVJ EC01144
SMOVL C01145 +MOVJ EC01145
SMOVL C01146 +MOVJ EC01146
SMOVL C01147 +MOVJ EC01147
SMOVL C01148 +MOVJ EC01148
SMOVL C01149 +MOVJ EC01149
SMOVL C01150 +MOVJ EC01150
SMOVL C01151 +MOVJ EC01151
SMOVL C01152 +MOVJ EC01152
SMOVL C01153 +MOVJ EC01153
SMOVL C01154 +MOVJ EC01154
SMOVL C01155 +MOVJ EC01155
SMOVL C01156 +MOVJ EC01156
SMOVL C01157 +MOVJ EC01157
SMOVL C01158 +MOVJ EC01158
SMOVL C01159 +MOVJ EC01159
SMOVL C01160 +MOVJ EC01160
SMOVL C01161 +MOVJ EC01161
SMOVL C01162 +MOVJ EC01162
SMOVL C01163 +MOVJ EC01163
SMOVL C01164 +MOVJ EC01164
SMOVL C01165 +MOVJ EC01165
SMOVL C01166 +MOVJ EC01166
SMOVL C01167 +MOVJ EC01167
SMOVL C01168 +MOVJ EC01168
SMOVL C01169 +MOVJ EC01169
SMOVL C01170 +MOVJ EC01170
SMOVL C01171 +MOVJ EC01171
SMOVL C01172 +MOVJ EC01172
SMOVL C01173 +MOVJ EC01173
SMOVL C01174 +MOVJ EC01174
SMOVL C01175 +MOVJ EC01175
SMOVL C01176 +MOVJ EC01176
SMOVL C01177 +MOVJ EC01177
SMOVL C01178 +MOVJ EC01178
SMOVL C01179 +MOVJ EC01179
SMOVL C01180 +MOVJ EC01180
SMOVL C01181 +MOVJ EC01181
SMOVL C01182 +MOVJ EC01182
SMOVL C01183 +MOVJ EC01183
SMOVL C01184 +MOVJ EC01184
SMOVL C01185 +MOVJ EC01185
SMOVL C01186 +MOVJ EC01186
SMOVL C01187 +MOVJ EC01187
SMOVL C01188 +MOVJ EC01188
SMOVL C01189 +MOVJ EC01189
SMOVL C01190 +MOVJ EC01190
SMOVL C01191 +MOVJ EC01191
SMOVL C01192 +MOVJ EC01192
SMOVL C01193 +MOVJ EC01193
SMOVL C01194 +MOVJ EC01194
SMOVL C01195 +MOVJ EC01195
SMOVL C01196 +MOVJ EC01196
SMOVL C01197 +MOVJ EC01197
SMOVL C01198 +MOVJ EC01198
SMOVL C01199 +MOVJ EC01199
SMOVL C01200 +MOVJ EC01200
SMOVL C01201 +MOVJ EC01201
SMOVL C01202 +MOVJ EC01202
SMOVL C01203 +MOVJ EC01203
SMOVL C01204 +MOVJ EC01204
SMOVL C01205 +MOVJ EC01205
SMOVL C01206 +MOVJ EC01206
SMOVL C01207 +MOVJ EC01207
SMOVL C01208 +MOVJ EC01208
SMOVL C01209 +MOVJ EC01209
SMOVL C01210 +MOVJ EC01210
SMOVL C01211 +MOVJ EC01211
SMOVL C01212 +MOVJ EC01212
SMOVL C01213 +MOVJ EC01213
SMOVL C01214 +MOVJ EC01214
SMOVL C01215 +MOVJ EC01215
SMOVL C01216 +MOVJ EC01216
SMOVL C01217 +MOVJ EC01217
SMOVL C01218 +MOVJ EC01218
SMOVL C01219 +MOVJ EC01219
SMOVL C01220 +MOVJ EC01220
SMOVL C01221 +MOVJ EC01221
SMOVL C01222 +MOVJ EC01222
SMOVL C01223 +MOVJ EC01223
SMOVL C01224 +MOVJ EC01224
SMOVL C01225 +MOVJ EC01225
SMOVL C01226 +MOVJ EC01226
SMOVL C01227 +MOVJ EC01227
SMOVL C01228 +MOVJ EC01228
SMOVL C01229 +MOVJ EC01229
SMOVL C01230 +MOVJ EC01230
SMOVL C01231 +MOVJ EC01231
SMOVL C01232 +MOVJ EC01232
SMOVL C01233 +MOVJ EC01233
SMOVL C01234 +MOVJ EC01234
SMOVL C01235 +MOVJ EC01235
SMOVL C01236 +MOVJ EC01236
SMOVL C01237 +MOVJ EC01237
SMOVL C01238 +MOVJ EC01238
SMOVL C01239 +MOVJ EC01239
SMOVL C01240 +MOVJ EC01240
SMOVL C01241 +MOVJ EC01241
SMOVL C01242 +MOVJ EC01242
SMOVL C01243 +MOVJ EC01243
SMOVL C01244 +MOVJ EC01244
SMOVL C01245 +MOVJ EC01245
SMOVL C01246 +MOVJ EC01246
SMOVL C01247 +MOVJ EC01247
SMOVL C01248 +MOVJ EC01248
SMOVL C01249 +MOVJ EC01249
SMOVL C01250 +MOVJ EC01250
SMOVL C01251 +MOVJ EC01251
SMOVL C01252 +MOVJ EC01252
SMOVL C01253 +MOVJ EC01253
SMOVL C01254 +MOVJ EC01254
SMOVL C01255 +MOVJ EC01255
SMOVL C01256 +MOVJ EC01256
SMOVL C01257 +MOVJ EC01257
SMOVL C01258 +MOVJ EC01258
SMOVL C01259 +MOVJ EC01259
SMOVL C01260 +MOVJ EC01260
SMOVL C01261 +MOVJ EC01261
SMOVL C01262 +MOVJ EC01262
SMOVL C01263 +MOVJ EC01263
SMOVL C01264 +MOVJ EC01264
SMOVL C01265 +MOVJ EC01265
SMOVL C01266 +MOVJ EC01266
SMOVL C01267 +MOVJ EC01267
SMOVL C01268 +MOVJ EC01268
SMOVL C01269 +MOVJ EC01269
SMOVL C01270 +MOVJ EC01270
SMOVL C01271 +MOVJ EC01271
SMOVL C01272 +MOVJ EC01272
SMOVL C01273 +MOVJ EC01273
SMOVL C01274 +MOVJ EC01274
SMOVL C01275 +MOVJ EC01275
SMOVL C01276 +MOVJ EC01276
SMOVL C01277 +MOVJ EC01277
SMOVL C01278 +MOVJ EC01278
SMOVL C01279 +MOVJ EC01279
SMOVL C01280 +MOVJ EC01280
SMOVL C01281 +MOVJ EC01281
SMOVL C01282 +MOVJ EC01282
SMOVL C01283 +MOVJ EC01283
SMOVL C01284 +MOVJ EC01284
SMOVL C01285 +MOVJ EC01285
SMOVL C01286 +MOVJ EC01286
SMOVL C01287 +MOVJ EC01287
SMOVL C01288 +MOVJ EC01288
SMOVL C01289 +MOVJ EC01289
SMOVL C01290 +MOVJ EC01290
SMOVL C01291 +MOVJ EC01291
SMOVL C01292 +MOVJ EC01292
SMOVL C01293 +MOVJ EC01293
SMOVL C01294 +MOVJ EC01294
SMOVL C01295 +MOVJ EC01295
SMOVL C01296 +MOVJ EC01296
SMOVL C01297 +MOVJ EC01297
SMOVL C01298 +MOVJ EC01298
SMOVL C01299 +MOVJ EC01299
